ABB RAPID module: qulvOK.mod

MODULE Module1

    CONST robtarget myPath0{255} := [
[[1351.7,1.5,938.01],[0.00139266,-0.491072,0.870802,-0.0234724],[0,-1,-1,0],[9E+09,9E+09,9E+09,9E+09,9E+09,9E+09]],
[[1348.2,2,938.01],[0.00139266,-0.491072,0.870802,-0.0234724],[0,-1,-1,0],[9E+09,9E+09,9E+09,9E+09,9E+09,9E+09]],
[[1346.2,3,938.01],[0.00139266,-0.491072,0.870802,-0.0234724],[0,-1,-1,0],[9E+09,9E+09,9E+09,9E+09,9E+09,9E+09]],
[[1345.7,3,938.01],[0.00139266,-0.491072,0.870802,-0.0234724],[0,-1,-1,0],[9E+09,9E+09,9E+09,9E+09,9E+09,9E+09]],
[[1342.7,5,938.01],[0.00139266,-0.491072,0.870802,-0.0234724],[0,-1,-1,0],[9E+09,9E+09,9E+09,9E+09,9E+09,9E+09]],
[[1340.2,3.5,938.01],[0.00139266,-0.491072,0.870802,-0.0234724],[0,-1,-1,0],[9E+09,9E+09,9E+09,9E+09,9E+09,9E+09]],
[[1339.2,2.5,938.01],[0.00139266,-0.491072,0.870802,-0.0234724],[0,-1,-1,0],[9E+09,9E+09,9E+09,9E+09,9E+09,9E+09]],
[[1336.2,2,938.01],[0.00139266,-0.491072,0.870802,-0.0234724],[0,-1,-1,0],[9E+09,9E+09,9E+09,9E+09,9E+09,9E+09]],
[[1335.7,1.5,938.01],[0.00139266,-0.491072,0.870802,-0.0234724],[0,-1,-1,0],[9E+09,9E+09,9E+09,9E+09,9E+09,9E+09]],
[[1327.7,2,938.01],[0.00139266,-0.491072,0.870802,-0.0234724],[0,-1,-1,0],[9E+09,9E+09,9E+09,9E+09,9E+09,9E+09]],
[[1327.2,2.5,938.01],[0.00139266,-0.491072,0.870802,-0.0234724],[0,-1,-1,0],[9E+09,9E+09,9E+09,9E+09,9E+09,9E+09]],
[[1326.7,2.5,938.01],[0.00139266,-0.491072,0.870802,-0.0234724],[0,-1,-1,0],[9E+09,9E+09,9E+09,9E+09,9E+09,9E+09]],
[[1326.2,3,938.01],[0.00139266,-0.491072,0.870802,-0.0234724],[0,-1,-1,0],[9E+09,9E+09,9E+09,9E+09,9E+09,9E+09]],
[[1319.7,6.5,938.01],[0.00139266,-0.491072,0.870802,-0.0234724],[0,-1,-1,0],[9E+09,9E+09,9E+09,9E+09,9E+09,9E+09]],
[[1319.7,6.5,938.01],[0.00139266,-0.491072,0.870802,-0.0234724],[0,-1,-1,0],[9E+09,9E+09,9E+09,9E+09,9E+09,9E+09]],
[[1319.7,6.5,938.01],[0.00139266,-0.491072,0.870802,-0.0234724],[0,-1,-1,0],[9E+09,9E+09,9E+09,9E+09,9E+09,9E+09]],
[[1319.2,7,938.01],[0.00139266,-0.491072,0.870802,-0.0234724],[0,-1,-1,0],[9E+09,9E+09,9E+09,9E+09,9E+09,9E+09]],
[[1310.2,14.5,938.01],[0.00139266,-0.491072,0.870802,-0.0234724],[0,-1,-1,0],[9E+09,9E+09,9E+09,9E+09,9E+09,9E+09]],
[[1310.2,14.5,938.01],[0.00139266,-0.491072,0.870802,-0.0234724],[0,-1,-1,0],[9E+09,9E+09,9E+09,9E+09,9E+09,9E+09]],
[[1310.2,14.5,938.01],[0.00139266,-0.491072,0.870802,-0.0234724],[0,-1,-1,0],[9E+09,9E+09,9E+09,9E+09,9E+09,9E+09]],
[[1310.2,14.5,938.01],[0.00139266,-0.491072,0.870802,-0.0234724],[0,-1,-1,0],[9E+09,9E+09,9E+09,9E+09,9E+09,9E+09]],
[[1307.2,18.5,938.01],[0.00139266,-0.491072,0.870802,-0.0234724],[0,-1,-1,0],[9E+09,9E+09,9E+09,9E+09,9E+09,9E+09]],
[[1303.7,23,938.01],[0.00139266,-0.491072,0.870802,-0.0234724],[0,-1,-1,0],[9E+09,9E+09,9E+09,9E+09,9E+09,9E+09]],
[[1303.7,22.5,938.01],[0.00139266,-0.491072,0.870802,-0.0234724],[0,-1,-1,0],[9E+09,9E+09,9E+09,9E+09,9E+09,9E+09]],
[[1302.2,25,938.01],[0.00139266,-0.491072,0.870802,-0.0234724],[0,-1,-1,0],[9E+09,9E+09,9E+09,9E+09,9E+09,9E+09]],
[[1302.2,25,938.01],[0.00139266,-0.491072,0.870802,-0.0234724],[0,-1,-1,0],[9E+09,9E+09,9E+09,9E+09,9E+09,9E+09]],
[[1301.7,25.5,938.01],[0.00139266,-0.491072,0.870802,-0.0234724],[0,-1,-1,0],[9E+09,9E+09,9E+09,9E+09,9E+09,9E+09]],
[[1301.7,25.5,938.01],[0.00139266,-0.491072,0.870802,-0.0234724],[0,-1,-1,0],[9E+09,9E+09,9E+09,9E+09,9E+09,9E+09]],
[[1299.7,28.5,938.01],[0.00139266,-0.491072,0.870802,-0.0234724],[0,-1,-1,0],[9E+09,9E+09,9E+09,9E+09,9E+09,9E+09]],
[[1299.7,28.5,938.01],[0.00139266,-0.491072,0.870802,-0.0234724],[0,-1,-1,0],[9E+09,9E+09,9E+09,9E+09,9E+09,9E+09]],
[[1298.7,30,938.01],[0.00139266,-0.491072,0.870802,-0.0234724],[0,-1,-1,0],[9E+09,9E+09,9E+09,9E+09,9E+09,9E+09]],
[[1298.7,30,938.01],[0.00139266,-0.491072,0.870802,-0.0234724],[0,-1,-1,0],[9E+09,9E+09,9E+09,9E+09,9E+09,9E+09]],
[[1297.2,32.5,938.01],[0.00139266,-0.491072,0.870802,-0.0234724],[0,-1,-1,0],[9E+09,9E+09,9E+09,9E+09,9E+09,9E+09]],
[[1295.2,36.5,938.01],[0.00139266,-0.491072,0.870802,-0.0234724],[0,-1,-1,0],[9E+09,9E+09,9E+09,9E+09,9E+09,9E+09]],
[[1295.2,36.5,938.01],[0.00139266,-0.491072,0.870802,-0.0234724],[0,-1,-1,0],[9E+09,9E+09,9E+09,9E+09,9E+09,9E+09]],
[[1294.2,39,938.01],[0.00139266,-0.491072,0.870802,-0.0234724],[0,-1,-1,0],[9E+09,9E+09,9E+09,9E+09,9E+09,9E+09]],
[[1293.7,40,938.01],[0.00139266,-0.491072,0.870802,-0.0234724],[0,-1,-1,0],[9E+09,9E+09,9E+09,9E+09,9E+09,9E+09]],
[[1293.2,41,938.01],[0.00139266,-0.491072,0.870802,-0.0234724],[0,-1,-1,0],[9E+09,9E+09,9E+09,9E+09,9E+09,9E+09]],
[[1293.2,41.5,938.01],[0.00139266,-0.491072,0.870802,-0.0234724],[0,-1,-1,0],[9E+09,9E+09,9E+09,9E+09,9E+09,9E+09]],
[[1292.7,42,938.01],[0.00139266,-0.491072,0.870802,-0.0234724],[0,-1,-1,0],[9E+09,9E+09,9E+09,9E+09,9E+09,9E+09]],
[[1292.7,42.5,938.01],[0.00139266,-0.491072,0.870802,-0.0234724],[0,-1,-1,0],[9E+09,9E+09,9E+09,9E+09,9E+09,9E+09]],
[[1292.7,42.5,938.01],[0.00139266,-0.491072,0.870802,-0.0234724],[0,-1,-1,0],[9E+09,9E+09,9E+09,9E+09,9E+09,9E+09]],
[[1293.2,57,938.01],[0.00139266,-0.491072,0.870802,-0.0234724],[0,-1,-1,0],[9E+09,9E+09,9E+09,9E+09,9E+09,9E+09]],
[[1293.7,58,938.01],[0.00139266,-0.491072,0.870802,-0.0234724],[0,-1,-1,0],[9E+09,9E+09,9E+09,9E+09,9E+09,9E+09]],
[[1293.7,58,938.01],[0.00139266,-0.491072,0.870802,-0.0234724],[0,-1,-1,0],[9E+09,9E+09,9E+09,9E+09,9E+09,9E+09]],
[[1295.7,61,938.01],[0.00139266,-0.491072,0.870802,-0.0234724],[0,-1,-1,0],[9E+09,9E+09,9E+09,9E+09,9E+09,9E+09]],
[[1296.7,62.5,938.01],[0.00139266,-0.491072,0.870802,-0.0234724],[0,-1,-1,0],[9E+09,9E+09,9E+09,9E+09,9E+09,9E+09]],
[[1302.2,67,938.01],[0.00139266,-0.491072,0.870802,-0.0234724],[0,-1,-1,0],[9E+09,9E+09,9E+09,9E+09,9E+09,9E+09]],
[[1302.2,67,938.01],[0.00139266,-0.491072,0.870802,-0.0234724],[0,-1,-1,0],[9E+09,9E+09,9E+09,9E+09,9E+09,9E+09]],
[[1304.2,68.5,938.01],[0.00139266,-0.491072,0.870802,-0.0234724],[0,-1,-1,0],[9E+09,9E+09,9E+09,9E+09,9E+09,9E+09]],
[[1305.2,69,938.01],[0.00139266,-0.491072,0.870802,-0.0234724],[0,-1,-1,0],[9E+09,9E+09,9E+09,9E+09,9E+09,9E+09]],
[[1305.2,69,938.01],[0.00139266,-0.491072,0.870802,-0.0234724],[0,-1,-1,0],[9E+09,9E+09,9E+09,9E+09,9E+09,9E+09]],
[[1307.2,70,938.01],[0.00139266,-0.491072,0.870802,-0.0234724],[0,-1,-1,0],[9E+09,9E+09,9E+09,9E+09,9E+09,9E+09]],
[[1308.7,70,938.01],[0.00139266,-0.491072,0.870802,-0.0234724],[0,-1,-1,0],[9E+09,9E+09,9E+09,9E+09,9E+09,9E+09]],
[[1310.2,72,938.01],[0.00139266,-0.491072,0.870802,-0.0234724],[0,-1,-1,0],[9E+09,9E+09,9E+09,9E+09,9E+09,9E+09]],
[[1313.7,71,938.01],[0.00139266,-0.491072,0.870802,-0.0234724],[0,-1,-1,0],[9E+09,9E+09,9E+09,9E+09,9E+09,9E+09]],
[[1314.2,71.5,938.01],[0.00139266,-0.491072,0.870802,-0.0234724],[0,-1,-1,0],[9E+09,9E+09,9E+09,9E+09,9E+09,9E+09]],
[[1317.7,72,938.01],[0.00139266,-0.491072,0.870802,-0.0234724],[0,-1,-1,0],[9E+09,9E+09,9E+09,9E+09,9E+09,9E+09]],
[[1317.7,72,938.01],[0.00139266,-0.491072,0.870802,-0.0234724],[0,-1,-1,0],[9E+09,9E+09,9E+09,9E+09,9E+09,9E+09]],
[[1317.7,72,938.01],[0.00139266,-0.491072,0.870802,-0.0234724],[0,-1,-1,0],[9E+09,9E+09,9E+09,9E+09,9E+09,9E+09]],
[[1310.2,72,938.01],[0.00139266,-0.491072,0.870802,-0.0234724],[0,-1,-1,0],[9E+09,9E+09,9E+09,9E+09,9E+09,9E+09]],
[[1307.7,73.5,938.01],[0.00139266,-0.491072,0.870802,-0.0234724],[0,-1,-1,0],[9E+09,9E+09,9E+09,9E+09,9E+09,9E+09]],
[[1301.2,74,938.01],[0.00139266,-0.491072,0.870802,-0.0234724],[0,-1,-1,0],[9E+09,9E+09,9E+09,9E+09,9E+09,9E+09]],
[[1300.7,74.5,938.01],[0.00139266,-0.491072,0.870802,-0.0234724],[0,-1,-1,0],[9E+09,9E+09,9E+09,9E+09,9E+09,9E+09]],
[[1299.7,74.5,938.01],[0.00139266,-0.491072,0.870802,-0.0234724],[0,-1,-1,0],[9E+09,9E+09,9E+09,9E+09,9E+09,9E+09]],
[[1299.2,75,938.01],[0.00139266,-0.491072,0.870802,-0.0234724],[0,-1,-1,0],[9E+09,9E+09,9E+09,9E+09,9E+09,9E+09]],
[[1295.7,76,938.01],[0.00139266,-0.491072,0.870802,-0.0234724],[0,-1,-1,0],[9E+09,9E+09,9E+09,9E+09,9E+09,9E+09]],
[[1295.7,76,938.01],[0.00139266,-0.491072,0.870802,-0.0234724],[0,-1,-1,0],[9E+09,9E+09,9E+09,9E+09,9E+09,9E+09]],
[[1295.2,76.5,938.01],[0.00139266,-0.491072,0.870802,-0.0234724],[0,-1,-1,0],[9E+09,9E+09,9E+09,9E+09,9E+09,9E+09]],
[[1294.2,76.5,938.01],[0.00139266,-0.491072,0.870802,-0.0234724],[0,-1,-1,0],[9E+09,9E+09,9E+09,9E+09,9E+09,9E+09]],
[[1292.7,77.5,938.01],[0.00139266,-0.491072,0.870802,-0.0234724],[0,-1,-1,0],[9E+09,9E+09,9E+09,9E+09,9E+09,9E+09]],
[[1292.2,77.5,938.01],[0.00139266,-0.491072,0.870802,-0.0234724],[0,-1,-1,0],[9E+09,9E+09,9E+09,9E+09,9E+09,9E+09]],
[[1292.2,77.5,938.01],[0.00139266,-0.491072,0.870802,-0.0234724],[0,-1,-1,0],[9E+09,9E+09,9E+09,9E+09,9E+09,9E+09]],
[[1286.7,80.5,938.01],[0.00139266,-0.491072,0.870802,-0.0234724],[0,-1,-1,0],[9E+09,9E+09,9E+09,9E+09,9E+09,9E+09]],
[[1286.7,80.5,938.01],[0.00139266,-0.491072,0.870802,-0.0234724],[0,-1,-1,0],[9E+09,9E+09,9E+09,9E+09,9E+09,9E+09]],
[[1286.7,80.5,938.01],[0.00139266,-0.491072,0.870802,-0.0234724],[0,-1,-1,0],[9E+09,9E+09,9E+09,9E+09,9E+09,9E+09]],
[[1280.7,75,938.01],[0.00139266,-0.491072,0.870802,-0.0234724],[0,-1,-1,0],[9E+09,9E+09,9E+09,9E+09,9E+09,9E+09]],
[[1281.2,68.5,938.01],[0.00139266,-0.491072,0.870802,-0.0234724],[0,-1,-1,0],[9E+09,9E+09,9E+09,9E+09,9E+09,9E+09]],
[[1281.2,68.5,938.01],[0.00139266,-0.491072,0.870802,-0.0234724],[0,-1,-1,0],[9E+09,9E+09,9E+09,9E+09,9E+09,9E+09]],
[[1282.7,66.5,938.01],[0.00139266,-0.491072,0.870802,-0.0234724],[0,-1,-1,0],[9E+09,9E+09,9E+09,9E+09,9E+09,9E+09]],
[[1282.7,66,938.01],[0.00139266,-0.491072,0.870802,-0.0234724],[0,-1,-1,0],[9E+09,9E+09,9E+09,9E+09,9E+09,9E+09]],
[[1280.7,63,938.01],[0.00139266,-0.491072,0.870802,-0.0234724],[0,-1,-1,0],[9E+09,9E+09,9E+09,9E+09,9E+09,9E+09]],
[[1280.2,63.5,938.01],[0.00139266,-0.491072,0.870802,-0.0234724],[0,-1,-1,0],[9E+09,9E+09,9E+09,9E+09,9E+09,9E+09]],
[[1279.7,63.5,938.01],[0.00139266,-0.491072,0.870802,-0.0234724],[0,-1,-1,0],[9E+09,9E+09,9E+09,9E+09,9E+09,9E+09]],
[[1278.2,64,938.01],[0.00139266,-0.491072,0.870802,-0.0234724],[0,-1,-1,0],[9E+09,9E+09,9E+09,9E+09,9E+09,9E+09]],
[[1277.7,64,938.01],[0.00139266,-0.491072,0.870802,-0.0234724],[0,-1,-1,0],[9E+09,9E+09,9E+09,9E+09,9E+09,9E+09]],
[[1276.7,64.5,938.01],[0.00139266,-0.491072,0.870802,-0.0234724],[0,-1,-1,0],[9E+09,9E+09,9E+09,9E+09,9E+09,9E+09]],
[[1276.2,64.5,938.01],[0.00139266,-0.491072,0.870802,-0.0234724],[0,-1,-1,0],[9E+09,9E+09,9E+09,9E+09,9E+09,9E+09]],
[[1275.7,65,938.01],[0.00139266,-0.491072,0.870802,-0.0234724],[0,-1,-1,0],[9E+09,9E+09,9E+09,9E+09,9E+09,9E+09]],
[[1275.7,65,938.01],[0.00139266,-0.491072,0.870802,-0.0234724],[0,-1,-1,0],[9E+09,9E+09,9E+09,9E+09,9E+09,9E+09]],
[[1274.2,66,938.01],[0.00139266,-0.491072,0.870802,-0.0234724],[0,-1,-1,0],[9E+09,9E+09,9E+09,9E+09,9E+09,9E+09]],
[[1273.2,66,938.01],[0.00139266,-0.491072,0.870802,-0.0234724],[0,-1,-1,0],[9E+09,9E+09,9E+09,9E+09,9E+09,9E+09]],
[[1266.2,74,938.01],[0.00139266,-0.491072,0.870802,-0.0234724],[0,-1,-1,0],[9E+09,9E+09,9E+09,9E+09,9E+09,9E+09]],
[[1266.2,74,938.01],[0.00139266,-0.491072,0.870802,-0.0234724],[0,-1,-1,0],[9E+09,9E+09,9E+09,9E+09,9E+09,9E+09]],
[[1266.2,74,938.01],[0.00139266,-0.491072,0.870802,-0.0234724],[0,-1,-1,0],[9E+09,9E+09,9E+09,9E+09,9E+09,9E+09]],
[[1266.2,74,938.01],[0.00139266,-0.491072,0.870802,-0.0234724],[0,-1,-1,0],[9E+09,9E+09,9E+09,9E+09,9E+09,9E+09]],
[[1266.2,74,938.01],[0.00139266,-0.491072,0.870802,-0.0234724],[0,-1,-1,0],[9E+09,9E+09,9E+09,9E+09,9E+09,9E+09]],
[[1266.2,84,938.01],[0.00139266,-0.491072,0.870802,-0.0234724],[0,-1,-1,0],[9E+09,9E+09,9E+09,9E+09,9E+09,9E+09]],
[[1266.7,85,938.01],[0.00139266,-0.491072,0.870802,-0.0234724],[0,-1,-1,0],[9E+09,9E+09,9E+09,9E+09,9E+09,9E+09]],
[[1270.7,88.5,938.01],[0.00139266,-0.491072,0.870802,-0.0234724],[0,-1,-1,0],[9E+09,9E+09,9E+09,9E+09,9E+09,9E+09]],
[[1274.7,89.5,938.01],[0.00139266,-0.491072,0.870802,-0.0234724],[0,-1,-1,0],[9E+09,9E+09,9E+09,9E+09,9E+09,9E+09]],
[[1275.2,90,938.01],[0.00139266,-0.491072,0.870802,-0.0234724],[0,-1,-1,0],[9E+09,9E+09,9E+09,9E+09,9E+09,9E+09]],
[[1279.2,92.5,938.01],[0.00139266,-0.491072,0.870802,-0.0234724],[0,-1,-1,0],[9E+09,9E+09,9E+09,9E+09,9E+09,9E+09]],
[[1278.7,93,938.01],[0.00139266,-0.491072,0.870802,-0.0234724],[0,-1,-1,0],[9E+09,9E+09,9E+09,9E+09,9E+09,9E+09]],
[[1278.7,94,938.01],[0.00139266,-0.491072,0.870802,-0.0234724],[0,-1,-1,0],[9E+09,9E+09,9E+09,9E+09,9E+09,9E+09]],
[[1278.2,94.5,938.01],[0.00139266,-0.491072,0.870802,-0.0234724],[0,-1,-1,0],[9E+09,9E+09,9E+09,9E+09,9E+09,9E+09]],
[[1278.7,106,938.01],[0.00139266,-0.491072,0.870802,-0.0234724],[0,-1,-1,0],[9E+09,9E+09,9E+09,9E+09,9E+09,9E+09]],
[[1279.2,108,938.01],[0.00139266,-0.491072,0.870802,-0.0234724],[0,-1,-1,0],[9E+09,9E+09,9E+09,9E+09,9E+09,9E+09]],
[[1279.7,109,938.01],[0.00139266,-0.491072,0.870802,-0.0234724],[0,-1,-1,0],[9E+09,9E+09,9E+09,9E+09,9E+09,9E+09]],
[[1280.2,110.5,938.01],[0.00139266,-0.491072,0.870802,-0.0234724],[0,-1,-1,0],[9E+09,9E+09,9E+09,9E+09,9E+09,9E+09]],
[[1280.2,110.5,938.01],[0.00139266,-0.491072,0.870802,-0.0234724],[0,-1,-1,0],[9E+09,9E+09,9E+09,9E+09,9E+09,9E+09]],
[[1280.7,111,938.01],[0.00139266,-0.491072,0.870802,-0.0234724],[0,-1,-1,0],[9E+09,9E+09,9E+09,9E+09,9E+09,9E+09]],
[[1280.7,111,938.01],[0.00139266,-0.491072,0.870802,-0.0234724],[0,-1,-1,0],[9E+09,9E+09,9E+09,9E+09,9E+09,9E+09]],
[[1285.7,117.5,938.01],[0.00139266,-0.491072,0.870802,-0.0234724],[0,-1,-1,0],[9E+09,9E+09,9E+09,9E+09,9E+09,9E+09]],
[[1285.7,118,938.01],[0.00139266,-0.491072,0.870802,-0.0234724],[0,-1,-1,0],[9E+09,9E+09,9E+09,9E+09,9E+09,9E+09]],
[[1286.2,118,938.01],[0.00139266,-0.491072,0.870802,-0.0234724],[0,-1,-1,0],[9E+09,9E+09,9E+09,9E+09,9E+09,9E+09]],
[[1287.2,119,938.01],[0.00139266,-0.491072,0.870802,-0.0234724],[0,-1,-1,0],[9E+09,9E+09,9E+09,9E+09,9E+09,9E+09]],
[[1288.2,119.5,938.01],[0.00139266,-0.491072,0.870802,-0.0234724],[0,-1,-1,0],[9E+09,9E+09,9E+09,9E+09,9E+09,9E+09]],
[[1290.2,120.5,938.01],[0.00139266,-0.491072,0.870802,-0.0234724],[0,-1,-1,0],[9E+09,9E+09,9E+09,9E+09,9E+09,9E+09]],
[[1291.7,121.5,938.01],[0.00139266,-0.491072,0.870802,-0.0234724],[0,-1,-1,0],[9E+09,9E+09,9E+09,9E+09,9E+09,9E+09]],
[[1292.2,121.5,938.01],[0.00139266,-0.491072,0.870802,-0.0234724],[0,-1,-1,0],[9E+09,9E+09,9E+09,9E+09,9E+09,9E+09]],
[[1292.2,121.5,938.01],[0.00139266,-0.491072,0.870802,-0.0234724],[0,-1,-1,0],[9E+09,9E+09,9E+09,9E+09,9E+09,9E+09]],
[[1301.2,121.5,938.01],[0.00139266,-0.491072,0.870802,-0.0234724],[0,-1,-1,0],[9E+09,9E+09,9E+09,9E+09,9E+09,9E+09]],
[[1301.7,121,938.01],[0.00139266,-0.491072,0.870802,-0.0234724],[0,-1,-1,0],[9E+09,9E+09,9E+09,9E+09,9E+09,9E+09]],
[[1302.7,121,938.01],[0.00139266,-0.491072,0.870802,-0.0234724],[0,-1,-1,0],[9E+09,9E+09,9E+09,9E+09,9E+09,9E+09]],
[[1303.2,120.5,938.01],[0.00139266,-0.491072,0.870802,-0.0234724],[0,-1,-1,0],[9E+09,9E+09,9E+09,9E+09,9E+09,9E+09]],
[[1306.2,119.5,938.01],[0.00139266,-0.491072,0.870802,-0.0234724],[0,-1,-1,0],[9E+09,9E+09,9E+09,9E+09,9E+09,9E+09]],
[[1306.2,119.5,938.01],[0.00139266,-0.491072,0.870802,-0.0234724],[0,-1,-1,0],[9E+09,9E+09,9E+09,9E+09,9E+09,9E+09]],
[[1308.7,119.5,938.01],[0.00139266,-0.491072,0.870802,-0.0234724],[0,-1,-1,0],[9E+09,9E+09,9E+09,9E+09,9E+09,9E+09]],
[[1309.2,119,938.01],[0.00139266,-0.491072,0.870802,-0.0234724],[0,-1,-1,0],[9E+09,9E+09,9E+09,9E+09,9E+09,9E+09]],
[[1310.7,119,938.01],[0.00139266,-0.491072,0.870802,-0.0234724],[0,-1,-1,0],[9E+09,9E+09,9E+09,9E+09,9E+09,9E+09]],
[[1311.2,118.5,938.01],[0.00139266,-0.491072,0.870802,-0.0234724],[0,-1,-1,0],[9E+09,9E+09,9E+09,9E+09,9E+09,9E+09]],
[[1311.7,118.5,938.01],[0.00139266,-0.491072,0.870802,-0.0234724],[0,-1,-1,0],[9E+09,9E+09,9E+09,9E+09,9E+09,9E+09]],
[[1312.7,117.5,938.01],[0.00139266,-0.491072,0.870802,-0.0234724],[0,-1,-1,0],[9E+09,9E+09,9E+09,9E+09,9E+09,9E+09]],
[[1312.7,116.5,938.01],[0.00139266,-0.491072,0.870802,-0.0234724],[0,-1,-1,0],[9E+09,9E+09,9E+09,9E+09,9E+09,9E+09]],
[[1312.2,116,938.01],[0.00139266,-0.491072,0.870802,-0.0234724],[0,-1,-1,0],[9E+09,9E+09,9E+09,9E+09,9E+09,9E+09]],
[[1312.2,115.5,938.01],[0.00139266,-0.491072,0.870802,-0.0234724],[0,-1,-1,0],[9E+09,9E+09,9E+09,9E+09,9E+09,9E+09]],
[[1311.7,115,938.01],[0.00139266,-0.491072,0.870802,-0.0234724],[0,-1,-1,0],[9E+09,9E+09,9E+09,9E+09,9E+09,9E+09]],
[[1311.7,114,938.01],[0.00139266,-0.491072,0.870802,-0.0234724],[0,-1,-1,0],[9E+09,9E+09,9E+09,9E+09,9E+09,9E+09]],
[[1312.2,113.5,938.01],[0.00139266,-0.491072,0.870802,-0.0234724],[0,-1,-1,0],[9E+09,9E+09,9E+09,9E+09,9E+09,9E+09]],
[[1313.2,113.5,938.01],[0.00139266,-0.491072,0.870802,-0.0234724],[0,-1,-1,0],[9E+09,9E+09,9E+09,9E+09,9E+09,9E+09]],
[[1313.7,114,938.01],[0.00139266,-0.491072,0.870802,-0.0234724],[0,-1,-1,0],[9E+09,9E+09,9E+09,9E+09,9E+09,9E+09]],
[[1320.2,114,938.01],[0.00139266,-0.491072,0.870802,-0.0234724],[0,-1,-1,0],[9E+09,9E+09,9E+09,9E+09,9E+09,9E+09]],
[[1325.2,120,938.01],[0.00139266,-0.491072,0.870802,-0.0234724],[0,-1,-1,0],[9E+09,9E+09,9E+09,9E+09,9E+09,9E+09]],
[[1325.2,120,938.01],[0.00139266,-0.491072,0.870802,-0.0234724],[0,-1,-1,0],[9E+09,9E+09,9E+09,9E+09,9E+09,9E+09]],
[[1326.2,120.5,938.01],[0.00139266,-0.491072,0.870802,-0.0234724],[0,-1,-1,0],[9E+09,9E+09,9E+09,9E+09,9E+09,9E+09]],
[[1341.2,121.5,938.01],[0.00139266,-0.491072,0.870802,-0.0234724],[0,-1,-1,0],[9E+09,9E+09,9E+09,9E+09,9E+09,9E+09]],
[[1341.7,121,938.01],[0.00139266,-0.491072,0.870802,-0.0234724],[0,-1,-1,0],[9E+09,9E+09,9E+09,9E+09,9E+09,9E+09]],
[[1342.7,121,938.01],[0.00139266,-0.491072,0.870802,-0.0234724],[0,-1,-1,0],[9E+09,9E+09,9E+09,9E+09,9E+09,9E+09]],
[[1343.2,120.5,938.01],[0.00139266,-0.491072,0.870802,-0.0234724],[0,-1,-1,0],[9E+09,9E+09,9E+09,9E+09,9E+09,9E+09]],
[[1343.7,113.5,938.01],[0.00139266,-0.491072,0.870802,-0.0234724],[0,-1,-1,0],[9E+09,9E+09,9E+09,9E+09,9E+09,9E+09]],
[[1343.7,113.5,938.01],[0.00139266,-0.491072,0.870802,-0.0234724],[0,-1,-1,0],[9E+09,9E+09,9E+09,9E+09,9E+09,9E+09]],
[[1343.7,113.5,938.01],[0.00139266,-0.491072,0.870802,-0.0234724],[0,-1,-1,0],[9E+09,9E+09,9E+09,9E+09,9E+09,9E+09]],
[[1343.7,113.5,938.01],[0.00139266,-0.491072,0.870802,-0.0234724],[0,-1,-1,0],[9E+09,9E+09,9E+09,9E+09,9E+09,9E+09]],
[[1346.7,113,938.01],[0.00139266,-0.491072,0.870802,-0.0234724],[0,-1,-1,0],[9E+09,9E+09,9E+09,9E+09,9E+09,9E+09]],
[[1347.2,112.5,938.01],[0.00139266,-0.491072,0.870802,-0.0234724],[0,-1,-1,0],[9E+09,9E+09,9E+09,9E+09,9E+09,9E+09]],
[[1348.7,112.5,938.01],[0.00139266,-0.491072,0.870802,-0.0234724],[0,-1,-1,0],[9E+09,9E+09,9E+09,9E+09,9E+09,9E+09]],
[[1349.2,112,938.01],[0.00139266,-0.491072,0.870802,-0.0234724],[0,-1,-1,0],[9E+09,9E+09,9E+09,9E+09,9E+09,9E+09]],
[[1352.7,111,938.01],[0.00139266,-0.491072,0.870802,-0.0234724],[0,-1,-1,0],[9E+09,9E+09,9E+09,9E+09,9E+09,9E+09]],
[[1352.7,111,938.01],[0.00139266,-0.491072,0.870802,-0.0234724],[0,-1,-1,0],[9E+09,9E+09,9E+09,9E+09,9E+09,9E+09]],
[[1352.7,111,938.01],[0.00139266,-0.491072,0.870802,-0.0234724],[0,-1,-1,0],[9E+09,9E+09,9E+09,9E+09,9E+09,9E+09]],
[[1356.7,108,938.01],[0.00139266,-0.491072,0.870802,-0.0234724],[0,-1,-1,0],[9E+09,9E+09,9E+09,9E+09,9E+09,9E+09]],
[[1356.2,105,938.01],[0.00139266,-0.491072,0.870802,-0.0234724],[0,-1,-1,0],[9E+09,9E+09,9E+09,9E+09,9E+09,9E+09]],
[[1356.2,105,938.01],[0.00139266,-0.491072,0.870802,-0.0234724],[0,-1,-1,0],[9E+09,9E+09,9E+09,9E+09,9E+09,9E+09]],
[[1353.2,102.5,938.01],[0.00139266,-0.491072,0.870802,-0.0234724],[0,-1,-1,0],[9E+09,9E+09,9E+09,9E+09,9E+09,9E+09]],
[[1353.2,102.5,938.01],[0.00139266,-0.491072,0.870802,-0.0234724],[0,-1,-1,0],[9E+09,9E+09,9E+09,9E+09,9E+09,9E+09]],
[[1353.2,102.5,938.01],[0.00139266,-0.491072,0.870802,-0.0234724],[0,-1,-1,0],[9E+09,9E+09,9E+09,9E+09,9E+09,9E+09]],
[[1352.7,99,938.01],[0.00139266,-0.491072,0.870802,-0.0234724],[0,-1,-1,0],[9E+09,9E+09,9E+09,9E+09,9E+09,9E+09]],
[[1352.2,98.5,938.01],[0.00139266,-0.491072,0.870802,-0.0234724],[0,-1,-1,0],[9E+09,9E+09,9E+09,9E+09,9E+09,9E+09]],
[[1352.2,97.5,938.01],[0.00139266,-0.491072,0.870802,-0.0234724],[0,-1,-1,0],[9E+09,9E+09,9E+09,9E+09,9E+09,9E+09]],
[[1350.7,95,938.01],[0.00139266,-0.491072,0.870802,-0.0234724],[0,-1,-1,0],[9E+09,9E+09,9E+09,9E+09,9E+09,9E+09]],
[[1350.7,95,938.01],[0.00139266,-0.491072,0.870802,-0.0234724],[0,-1,-1,0],[9E+09,9E+09,9E+09,9E+09,9E+09,9E+09]],
[[1350.7,95,938.01],[0.00139266,-0.491072,0.870802,-0.0234724],[0,-1,-1,0],[9E+09,9E+09,9E+09,9E+09,9E+09,9E+09]],
[[1352.2,89,938.01],[0.00139266,-0.491072,0.870802,-0.0234724],[0,-1,-1,0],[9E+09,9E+09,9E+09,9E+09,9E+09,9E+09]],
[[1350.7,86.5,938.01],[0.00139266,-0.491072,0.870802,-0.0234724],[0,-1,-1,0],[9E+09,9E+09,9E+09,9E+09,9E+09,9E+09]],
[[1352.7,83.5,938.01],[0.00139266,-0.491072,0.870802,-0.0234724],[0,-1,-1,0],[9E+09,9E+09,9E+09,9E+09,9E+09,9E+09]],
[[1353.7,81,938.01],[0.00139266,-0.491072,0.870802,-0.0234724],[0,-1,-1,0],[9E+09,9E+09,9E+09,9E+09,9E+09,9E+09]],
[[1353.7,81,938.01],[0.00139266,-0.491072,0.870802,-0.0234724],[0,-1,-1,0],[9E+09,9E+09,9E+09,9E+09,9E+09,9E+09]],
[[1368.2,78.5,938.01],[0.00139266,-0.491072,0.870802,-0.0234724],[0,-1,-1,0],[9E+09,9E+09,9E+09,9E+09,9E+09,9E+09]],
[[1368.2,78.5,938.01],[0.00139266,-0.491072,0.870802,-0.0234724],[0,-1,-1,0],[9E+09,9E+09,9E+09,9E+09,9E+09,9E+09]],
[[1368.2,78.5,938.01],[0.00139266,-0.491072,0.870802,-0.0234724],[0,-1,-1,0],[9E+09,9E+09,9E+09,9E+09,9E+09,9E+09]],
[[1368.2,78.5,938.01],[0.00139266,-0.491072,0.870802,-0.0234724],[0,-1,-1,0],[9E+09,9E+09,9E+09,9E+09,9E+09,9E+09]],
[[1368.2,78,938.01],[0.00139266,-0.491072,0.870802,-0.0234724],[0,-1,-1,0],[9E+09,9E+09,9E+09,9E+09,9E+09,9E+09]],
[[1370.2,77.5,938.01],[0.00139266,-0.491072,0.870802,-0.0234724],[0,-1,-1,0],[9E+09,9E+09,9E+09,9E+09,9E+09,9E+09]],
[[1371.2,77.5,938.01],[0.00139266,-0.491072,0.870802,-0.0234724],[0,-1,-1,0],[9E+09,9E+09,9E+09,9E+09,9E+09,9E+09]],
[[1371.7,77,938.01],[0.00139266,-0.491072,0.870802,-0.0234724],[0,-1,-1,0],[9E+09,9E+09,9E+09,9E+09,9E+09,9E+09]],
[[1372.2,77,938.01],[0.00139266,-0.491072,0.870802,-0.0234724],[0,-1,-1,0],[9E+09,9E+09,9E+09,9E+09,9E+09,9E+09]],
[[1373.7,76.5,938.01],[0.00139266,-0.491072,0.870802,-0.0234724],[0,-1,-1,0],[9E+09,9E+09,9E+09,9E+09,9E+09,9E+09]],
[[1374.2,76.5,938.01],[0.00139266,-0.491072,0.870802,-0.0234724],[0,-1,-1,0],[9E+09,9E+09,9E+09,9E+09,9E+09,9E+09]],
[[1374.7,76,938.01],[0.00139266,-0.491072,0.870802,-0.0234724],[0,-1,-1,0],[9E+09,9E+09,9E+09,9E+09,9E+09,9E+09]],
[[1375.2,76,938.01],[0.00139266,-0.491072,0.870802,-0.0234724],[0,-1,-1,0],[9E+09,9E+09,9E+09,9E+09,9E+09,9E+09]],
[[1375.7,76,938.01],[0.00139266,-0.491072,0.870802,-0.0234724],[0,-1,-1,0],[9E+09,9E+09,9E+09,9E+09,9E+09,9E+09]],
[[1376.2,75.5,938.01],[0.00139266,-0.491072,0.870802,-0.0234724],[0,-1,-1,0],[9E+09,9E+09,9E+09,9E+09,9E+09,9E+09]],
[[1377.2,75,938.01],[0.00139266,-0.491072,0.870802,-0.0234724],[0,-1,-1,0],[9E+09,9E+09,9E+09,9E+09,9E+09,9E+09]],
[[1377.2,75,938.01],[0.00139266,-0.491072,0.870802,-0.0234724],[0,-1,-1,0],[9E+09,9E+09,9E+09,9E+09,9E+09,9E+09]],
[[1379.2,74,938.01],[0.00139266,-0.491072,0.870802,-0.0234724],[0,-1,-1,0],[9E+09,9E+09,9E+09,9E+09,9E+09,9E+09]],
[[1379.2,74,938.01],[0.00139266,-0.491072,0.870802,-0.0234724],[0,-1,-1,0],[9E+09,9E+09,9E+09,9E+09,9E+09,9E+09]],
[[1381.7,72.5,938.01],[0.00139266,-0.491072,0.870802,-0.0234724],[0,-1,-1,0],[9E+09,9E+09,9E+09,9E+09,9E+09,9E+09]],
[[1384.2,71,938.01],[0.00139266,-0.491072,0.870802,-0.0234724],[0,-1,-1,0],[9E+09,9E+09,9E+09,9E+09,9E+09,9E+09]],
[[1384.2,71,938.01],[0.00139266,-0.491072,0.870802,-0.0234724],[0,-1,-1,0],[9E+09,9E+09,9E+09,9E+09,9E+09,9E+09]],
[[1384.2,71,938.01],[0.00139266,-0.491072,0.870802,-0.0234724],[0,-1,-1,0],[9E+09,9E+09,9E+09,9E+09,9E+09,9E+09]],
[[1384.2,71,938.01],[0.00139266,-0.491072,0.870802,-0.0234724],[0,-1,-1,0],[9E+09,9E+09,9E+09,9E+09,9E+09,9E+09]],
[[1385.2,70.5,938.01],[0.00139266,-0.491072,0.870802,-0.0234724],[0,-1,-1,0],[9E+09,9E+09,9E+09,9E+09,9E+09,9E+09]],
[[1386.2,69.5,938.01],[0.00139266,-0.491072,0.870802,-0.0234724],[0,-1,-1,0],[9E+09,9E+09,9E+09,9E+09,9E+09,9E+09]],
[[1388.7,67.5,938.01],[0.00139266,-0.491072,0.870802,-0.0234724],[0,-1,-1,0],[9E+09,9E+09,9E+09,9E+09,9E+09,9E+09]],
[[1392.7,63.5,938.01],[0.00139266,-0.491072,0.870802,-0.0234724],[0,-1,-1,0],[9E+09,9E+09,9E+09,9E+09,9E+09,9E+09]],
[[1393.2,63,938.01],[0.00139266,-0.491072,0.870802,-0.0234724],[0,-1,-1,0],[9E+09,9E+09,9E+09,9E+09,9E+09,9E+09]],
[[1395.2,60,938.01],[0.00139266,-0.491072,0.870802,-0.0234724],[0,-1,-1,0],[9E+09,9E+09,9E+09,9E+09,9E+09,9E+09]],
[[1395.7,59,938.01],[0.00139266,-0.491072,0.870802,-0.0234724],[0,-1,-1,0],[9E+09,9E+09,9E+09,9E+09,9E+09,9E+09]],
[[1396.2,58.5,938.01],[0.00139266,-0.491072,0.870802,-0.0234724],[0,-1,-1,0],[9E+09,9E+09,9E+09,9E+09,9E+09,9E+09]],
[[1396.7,57.5,938.01],[0.00139266,-0.491072,0.870802,-0.0234724],[0,-1,-1,0],[9E+09,9E+09,9E+09,9E+09,9E+09,9E+09]],
[[1397.2,56.5,938.01],[0.00139266,-0.491072,0.870802,-0.0234724],[0,-1,-1,0],[9E+09,9E+09,9E+09,9E+09,9E+09,9E+09]],
[[1397.7,56,938.01],[0.00139266,-0.491072,0.870802,-0.0234724],[0,-1,-1,0],[9E+09,9E+09,9E+09,9E+09,9E+09,9E+09]],
[[1397.7,56,938.01],[0.00139266,-0.491072,0.870802,-0.0234724],[0,-1,-1,0],[9E+09,9E+09,9E+09,9E+09,9E+09,9E+09]],
[[1398.2,52.5,938.01],[0.00139266,-0.491072,0.870802,-0.0234724],[0,-1,-1,0],[9E+09,9E+09,9E+09,9E+09,9E+09,9E+09]],
[[1398.7,51,938.01],[0.00139266,-0.491072,0.870802,-0.0234724],[0,-1,-1,0],[9E+09,9E+09,9E+09,9E+09,9E+09,9E+09]],
[[1397.7,44.5,938.01],[0.00139266,-0.491072,0.870802,-0.0234724],[0,-1,-1,0],[9E+09,9E+09,9E+09,9E+09,9E+09,9E+09]],
[[1397.7,44.5,938.01],[0.00139266,-0.491072,0.870802,-0.0234724],[0,-1,-1,0],[9E+09,9E+09,9E+09,9E+09,9E+09,9E+09]],
[[1397.7,44.5,938.01],[0.00139266,-0.491072,0.870802,-0.0234724],[0,-1,-1,0],[9E+09,9E+09,9E+09,9E+09,9E+09,9E+09]],
[[1400.7,42.5,938.01],[0.00139266,-0.491072,0.870802,-0.0234724],[0,-1,-1,0],[9E+09,9E+09,9E+09,9E+09,9E+09,9E+09]],
[[1400.7,42.5,938.01],[0.00139266,-0.491072,0.870802,-0.0234724],[0,-1,-1,0],[9E+09,9E+09,9E+09,9E+09,9E+09,9E+09]],
[[1401.2,41.5,938.01],[0.00139266,-0.491072,0.870802,-0.0234724],[0,-1,-1,0],[9E+09,9E+09,9E+09,9E+09,9E+09,9E+09]],
[[1401.2,35.5,938.01],[0.00139266,-0.491072,0.870802,-0.0234724],[0,-1,-1,0],[9E+09,9E+09,9E+09,9E+09,9E+09,9E+09]],
[[1401.2,35.5,938.01],[0.00139266,-0.491072,0.870802,-0.0234724],[0,-1,-1,0],[9E+09,9E+09,9E+09,9E+09,9E+09,9E+09]],
[[1400.7,34.5,938.01],[0.00139266,-0.491072,0.870802,-0.0234724],[0,-1,-1,0],[9E+09,9E+09,9E+09,9E+09,9E+09,9E+09]],
[[1396.7,31.5,938.01],[0.00139266,-0.491072,0.870802,-0.0234724],[0,-1,-1,0],[9E+09,9E+09,9E+09,9E+09,9E+09,9E+09]],
[[1396.7,31.5,938.01],[0.00139266,-0.491072,0.870802,-0.0234724],[0,-1,-1,0],[9E+09,9E+09,9E+09,9E+09,9E+09,9E+09]],
[[1396.7,31.5,938.01],[0.00139266,-0.491072,0.870802,-0.0234724],[0,-1,-1,0],[9E+09,9E+09,9E+09,9E+09,9E+09,9E+09]],
[[1396.2,31.5,938.01],[0.00139266,-0.491072,0.870802,-0.0234724],[0,-1,-1,0],[9E+09,9E+09,9E+09,9E+09,9E+09,9E+09]],
[[1396.2,31.5,938.01],[0.00139266,-0.491072,0.870802,-0.0234724],[0,-1,-1,0],[9E+09,9E+09,9E+09,9E+09,9E+09,9E+09]],
[[1390.2,30.5,938.01],[0.00139266,-0.491072,0.870802,-0.0234724],[0,-1,-1,0],[9E+09,9E+09,9E+09,9E+09,9E+09,9E+09]],
[[1390.2,30.5,938.01],[0.00139266,-0.491072,0.870802,-0.0234724],[0,-1,-1,0],[9E+09,9E+09,9E+09,9E+09,9E+09,9E+09]],
[[1385.2,25,938.01],[0.00139266,-0.491072,0.870802,-0.0234724],[0,-1,-1,0],[9E+09,9E+09,9E+09,9E+09,9E+09,9E+09]],
[[1384.7,24.5,938.01],[0.00139266,-0.491072,0.870802,-0.0234724],[0,-1,-1,0],[9E+09,9E+09,9E+09,9E+09,9E+09,9E+09]],
[[1384.7,24.5,938.01],[0.00139266,-0.491072,0.870802,-0.0234724],[0,-1,-1,0],[9E+09,9E+09,9E+09,9E+09,9E+09,9E+09]],
[[1384.2,24,938.01],[0.00139266,-0.491072,0.870802,-0.0234724],[0,-1,-1,0],[9E+09,9E+09,9E+09,9E+09,9E+09,9E+09]],
[[1381.7,20.5,938.01],[0.00139266,-0.491072,0.870802,-0.0234724],[0,-1,-1,0],[9E+09,9E+09,9E+09,9E+09,9E+09,9E+09]],
[[1381.2,19.5,938.01],[0.00139266,-0.491072,0.870802,-0.0234724],[0,-1,-1,0],[9E+09,9E+09,9E+09,9E+09,9E+09,9E+09]],
[[1380.7,19,938.01],[0.00139266,-0.491072,0.870802,-0.0234724],[0,-1,-1,0],[9E+09,9E+09,9E+09,9E+09,9E+09,9E+09]],
[[1380.7,19,938.01],[0.00139266,-0.491072,0.870802,-0.0234724],[0,-1,-1,0],[9E+09,9E+09,9E+09,9E+09,9E+09,9E+09]],
[[1377.7,15,938.01],[0.00139266,-0.491072,0.870802,-0.0234724],[0,-1,-1,0],[9E+09,9E+09,9E+09,9E+09,9E+09,9E+09]],
[[1376.7,13.5,938.01],[0.00139266,-0.491072,0.870802,-0.0234724],[0,-1,-1,0],[9E+09,9E+09,9E+09,9E+09,9E+09,9E+09]],
[[1371.2,7.5,938.01],[0.00139266,-0.491072,0.870802,-0.0234724],[0,-1,-1,0],[9E+09,9E+09,9E+09,9E+09,9E+09,9E+09]],
[[1370.7,7.5,938.01],[0.00139266,-0.491072,0.870802,-0.0234724],[0,-1,-1,0],[9E+09,9E+09,9E+09,9E+09,9E+09,9E+09]],
[[1367.2,5,938.01],[0.00139266,-0.491072,0.870802,-0.0234724],[0,-1,-1,0],[9E+09,9E+09,9E+09,9E+09,9E+09,9E+09]],
[[1367.2,5,938.01],[0.00139266,-0.491072,0.870802,-0.0234724],[0,-1,-1,0],[9E+09,9E+09,9E+09,9E+09,9E+09,9E+09]],
[[1366.7,4.5,938.01],[0.00139266,-0.491072,0.870802,-0.0234724],[0,-1,-1,0],[9E+09,9E+09,9E+09,9E+09,9E+09,9E+09]],
[[1366.2,4.5,938.01],[0.00139266,-0.491072,0.870802,-0.0234724],[0,-1,-1,0],[9E+09,9E+09,9E+09,9E+09,9E+09,9E+09]],
[[1365.2,4,938.01],[0.00139266,-0.491072,0.870802,-0.0234724],[0,-1,-1,0],[9E+09,9E+09,9E+09,9E+09,9E+09,9E+09]],
[[1364.7,3.5,938.01],[0.00139266,-0.491072,0.870802,-0.0234724],[0,-1,-1,0],[9E+09,9E+09,9E+09,9E+09,9E+09,9E+09]],
[[1363.7,3,938.01],[0.00139266,-0.491072,0.870802,-0.0234724],[0,-1,-1,0],[9E+09,9E+09,9E+09,9E+09,9E+09,9E+09]],
[[1362.7,2.5,938.01],[0.00139266,-0.491072,0.870802,-0.0234724],[0,-1,-1,0],[9E+09,9E+09,9E+09,9E+09,9E+09,9E+09]],
[[1361.7,2,938.01],[0.00139266,-0.491072,0.870802,-0.0234724],[0,-1,-1,0],[9E+09,9E+09,9E+09,9E+09,9E+09,9E+09]],
[[1358.2,1.5,938.01],[0.00139266,-0.491072,0.870802,-0.0234724],[0,-1,-1,0],[9E+09,9E+09,9E+09,9E+09,9E+09,9E+09]],
[[1358.7,1.5,938.01],[0.00139266,-0.491072,0.870802,-0.0234724],[0,-1,-1,0],[9E+09,9E+09,9E+09,9E+09,9E+09,9E+09]]
];
CONST robtarget myPath1{15} := [
[[1311.7,115,938.01],[0.00139266,-0.491072,0.870802,-0.0234724],[0,-1,-1,0],[9E+09,9E+09,9E+09,9E+09,9E+09,9E+09]],
[[1312.2,115.5,938.01],[0.00139266,-0.491072,0.870802,-0.0234724],[0,-1,-1,0],[9E+09,9E+09,9E+09,9E+09,9E+09,9E+09]],
[[1312.2,116,938.01],[0.00139266,-0.491072,0.870802,-0.0234724],[0,-1,-1,0],[9E+09,9E+09,9E+09,9E+09,9E+09,9E+09]],
[[1312.7,116.5,938.01],[0.00139266,-0.491072,0.870802,-0.0234724],[0,-1,-1,0],[9E+09,9E+09,9E+09,9E+09,9E+09,9E+09]],
[[1312.7,117.5,938.01],[0.00139266,-0.491072,0.870802,-0.0234724],[0,-1,-1,0],[9E+09,9E+09,9E+09,9E+09,9E+09,9E+09]],
[[1311.7,118.5,938.01],[0.00139266,-0.491072,0.870802,-0.0234724],[0,-1,-1,0],[9E+09,9E+09,9E+09,9E+09,9E+09,9E+09]],
[[1310.7,118.5,938.01],[0.00139266,-0.491072,0.870802,-0.0234724],[0,-1,-1,0],[9E+09,9E+09,9E+09,9E+09,9E+09,9E+09]],
[[1310.2,119,938.01],[0.00139266,-0.491072,0.870802,-0.0234724],[0,-1,-1,0],[9E+09,9E+09,9E+09,9E+09,9E+09,9E+09]],
[[1309.2,119,938.01],[0.00139266,-0.491072,0.870802,-0.0234724],[0,-1,-1,0],[9E+09,9E+09,9E+09,9E+09,9E+09,9E+09]],
[[1308.7,119.5,938.01],[0.00139266,-0.491072,0.870802,-0.0234724],[0,-1,-1,0],[9E+09,9E+09,9E+09,9E+09,9E+09,9E+09]],
[[1306.2,119.5,938.01],[0.00139266,-0.491072,0.870802,-0.0234724],[0,-1,-1,0],[9E+09,9E+09,9E+09,9E+09,9E+09,9E+09]],
[[1306.2,116.5,938.01],[0.00139266,-0.491072,0.870802,-0.0234724],[0,-1,-1,0],[9E+09,9E+09,9E+09,9E+09,9E+09,9E+09]],
[[1306.7,116,938.01],[0.00139266,-0.491072,0.870802,-0.0234724],[0,-1,-1,0],[9E+09,9E+09,9E+09,9E+09,9E+09,9E+09]],
[[1306.7,115.5,938.01],[0.00139266,-0.491072,0.870802,-0.0234724],[0,-1,-1,0],[9E+09,9E+09,9E+09,9E+09,9E+09,9E+09]],
[[1307.2,115,938.01],[0.00139266,-0.491072,0.870802,-0.0234724],[0,-1,-1,0],[9E+09,9E+09,9E+09,9E+09,9E+09,9E+09]]
];
CONST robtarget myPath2{6} := [
[[1350.7,86.5,938.01],[0.00139266,-0.491072,0.870802,-0.0234724],[0,-1,-1,0],[9E+09,9E+09,9E+09,9E+09,9E+09,9E+09]],
[[1352.2,89,938.01],[0.00139266,-0.491072,0.870802,-0.0234724],[0,-1,-1,0],[9E+09,9E+09,9E+09,9E+09,9E+09,9E+09]],
[[1350.7,95,938.01],[0.00139266,-0.491072,0.870802,-0.0234724],[0,-1,-1,0],[9E+09,9E+09,9E+09,9E+09,9E+09,9E+09]],
[[1348.2,95.5,938.01],[0.00139266,-0.491072,0.870802,-0.0234724],[0,-1,-1,0],[9E+09,9E+09,9E+09,9E+09,9E+09,9E+09]],
[[1345.2,95,938.01],[0.00139266,-0.491072,0.870802,-0.0234724],[0,-1,-1,0],[9E+09,9E+09,9E+09,9E+09,9E+09,9E+09]],
[[1342.2,92.5,938.01],[0.00139266,-0.491072,0.870802,-0.0234724],[0,-1,-1,0],[9E+09,9E+09,9E+09,9E+09,9E+09,9E+09]]
];
CONST robtarget myPath3{146} := [
[[1310.2,72,938.01],[0.00139266,-0.491072,0.870802,-0.0234724],[0,-1,-1,0],[9E+09,9E+09,9E+09,9E+09,9E+09,9E+09]],
[[1317.7,72,938.01],[0.00139266,-0.491072,0.870802,-0.0234724],[0,-1,-1,0],[9E+09,9E+09,9E+09,9E+09,9E+09,9E+09]],
[[1318.2,74.5,938.01],[0.00139266,-0.491072,0.870802,-0.0234724],[0,-1,-1,0],[9E+09,9E+09,9E+09,9E+09,9E+09,9E+09]],
[[1318.7,75,938.01],[0.00139266,-0.491072,0.870802,-0.0234724],[0,-1,-1,0],[9E+09,9E+09,9E+09,9E+09,9E+09,9E+09]],
[[1318.7,75.5,938.01],[0.00139266,-0.491072,0.870802,-0.0234724],[0,-1,-1,0],[9E+09,9E+09,9E+09,9E+09,9E+09,9E+09]],
[[1319.2,76,938.01],[0.00139266,-0.491072,0.870802,-0.0234724],[0,-1,-1,0],[9E+09,9E+09,9E+09,9E+09,9E+09,9E+09]],
[[1319.2,76.5,938.01],[0.00139266,-0.491072,0.870802,-0.0234724],[0,-1,-1,0],[9E+09,9E+09,9E+09,9E+09,9E+09,9E+09]],
[[1319.7,77,938.01],[0.00139266,-0.491072,0.870802,-0.0234724],[0,-1,-1,0],[9E+09,9E+09,9E+09,9E+09,9E+09,9E+09]],
[[1320.2,78.5,938.01],[0.00139266,-0.491072,0.870802,-0.0234724],[0,-1,-1,0],[9E+09,9E+09,9E+09,9E+09,9E+09,9E+09]],
[[1325.7,83,938.01],[0.00139266,-0.491072,0.870802,-0.0234724],[0,-1,-1,0],[9E+09,9E+09,9E+09,9E+09,9E+09,9E+09]],
[[1325.7,83,938.01],[0.00139266,-0.491072,0.870802,-0.0234724],[0,-1,-1,0],[9E+09,9E+09,9E+09,9E+09,9E+09,9E+09]],
[[1326.2,83.5,938.01],[0.00139266,-0.491072,0.870802,-0.0234724],[0,-1,-1,0],[9E+09,9E+09,9E+09,9E+09,9E+09,9E+09]],
[[1326.2,83.5,938.01],[0.00139266,-0.491072,0.870802,-0.0234724],[0,-1,-1,0],[9E+09,9E+09,9E+09,9E+09,9E+09,9E+09]],
[[1330.2,85.5,938.01],[0.00139266,-0.491072,0.870802,-0.0234724],[0,-1,-1,0],[9E+09,9E+09,9E+09,9E+09,9E+09,9E+09]],
[[1330.2,85.5,938.01],[0.00139266,-0.491072,0.870802,-0.0234724],[0,-1,-1,0],[9E+09,9E+09,9E+09,9E+09,9E+09,9E+09]],
[[1330.2,85.5,938.01],[0.00139266,-0.491072,0.870802,-0.0234724],[0,-1,-1,0],[9E+09,9E+09,9E+09,9E+09,9E+09,9E+09]],
[[1330.2,85.5,938.01],[0.00139266,-0.491072,0.870802,-0.0234724],[0,-1,-1,0],[9E+09,9E+09,9E+09,9E+09,9E+09,9E+09]],
[[1331.2,86,938.01],[0.00139266,-0.491072,0.870802,-0.0234724],[0,-1,-1,0],[9E+09,9E+09,9E+09,9E+09,9E+09,9E+09]],
[[1331.2,86,938.01],[0.00139266,-0.491072,0.870802,-0.0234724],[0,-1,-1,0],[9E+09,9E+09,9E+09,9E+09,9E+09,9E+09]],
[[1336.2,88,938.01],[0.00139266,-0.491072,0.870802,-0.0234724],[0,-1,-1,0],[9E+09,9E+09,9E+09,9E+09,9E+09,9E+09]],
[[1336.2,88,938.01],[0.00139266,-0.491072,0.870802,-0.0234724],[0,-1,-1,0],[9E+09,9E+09,9E+09,9E+09,9E+09,9E+09]],
[[1336.2,88,938.01],[0.00139266,-0.491072,0.870802,-0.0234724],[0,-1,-1,0],[9E+09,9E+09,9E+09,9E+09,9E+09,9E+09]],
[[1342.2,89,938.01],[0.00139266,-0.491072,0.870802,-0.0234724],[0,-1,-1,0],[9E+09,9E+09,9E+09,9E+09,9E+09,9E+09]],
[[1342.2,89,938.01],[0.00139266,-0.491072,0.870802,-0.0234724],[0,-1,-1,0],[9E+09,9E+09,9E+09,9E+09,9E+09,9E+09]],
[[1342.2,92.5,938.01],[0.00139266,-0.491072,0.870802,-0.0234724],[0,-1,-1,0],[9E+09,9E+09,9E+09,9E+09,9E+09,9E+09]],
[[1345.2,95,938.01],[0.00139266,-0.491072,0.870802,-0.0234724],[0,-1,-1,0],[9E+09,9E+09,9E+09,9E+09,9E+09,9E+09]],
[[1348.2,95.5,938.01],[0.00139266,-0.491072,0.870802,-0.0234724],[0,-1,-1,0],[9E+09,9E+09,9E+09,9E+09,9E+09,9E+09]],
[[1350.7,95,938.01],[0.00139266,-0.491072,0.870802,-0.0234724],[0,-1,-1,0],[9E+09,9E+09,9E+09,9E+09,9E+09,9E+09]],
[[1352.2,97.5,938.01],[0.00139266,-0.491072,0.870802,-0.0234724],[0,-1,-1,0],[9E+09,9E+09,9E+09,9E+09,9E+09,9E+09]],
[[1352.2,98.5,938.01],[0.00139266,-0.491072,0.870802,-0.0234724],[0,-1,-1,0],[9E+09,9E+09,9E+09,9E+09,9E+09,9E+09]],
[[1352.7,99,938.01],[0.00139266,-0.491072,0.870802,-0.0234724],[0,-1,-1,0],[9E+09,9E+09,9E+09,9E+09,9E+09,9E+09]],
[[1353.2,102.5,938.01],[0.00139266,-0.491072,0.870802,-0.0234724],[0,-1,-1,0],[9E+09,9E+09,9E+09,9E+09,9E+09,9E+09]],
[[1353.2,102.5,938.01],[0.00139266,-0.491072,0.870802,-0.0234724],[0,-1,-1,0],[9E+09,9E+09,9E+09,9E+09,9E+09,9E+09]],
[[1353.2,102.5,938.01],[0.00139266,-0.491072,0.870802,-0.0234724],[0,-1,-1,0],[9E+09,9E+09,9E+09,9E+09,9E+09,9E+09]],
[[1353.2,102.5,938.01],[0.00139266,-0.491072,0.870802,-0.0234724],[0,-1,-1,0],[9E+09,9E+09,9E+09,9E+09,9E+09,9E+09]],
[[1356.2,105,938.01],[0.00139266,-0.491072,0.870802,-0.0234724],[0,-1,-1,0],[9E+09,9E+09,9E+09,9E+09,9E+09,9E+09]],
[[1356.7,108,938.01],[0.00139266,-0.491072,0.870802,-0.0234724],[0,-1,-1,0],[9E+09,9E+09,9E+09,9E+09,9E+09,9E+09]],
[[1352.7,111,938.01],[0.00139266,-0.491072,0.870802,-0.0234724],[0,-1,-1,0],[9E+09,9E+09,9E+09,9E+09,9E+09,9E+09]],
[[1352.7,111,938.01],[0.00139266,-0.491072,0.870802,-0.0234724],[0,-1,-1,0],[9E+09,9E+09,9E+09,9E+09,9E+09,9E+09]],
[[1352.7,111,938.01],[0.00139266,-0.491072,0.870802,-0.0234724],[0,-1,-1,0],[9E+09,9E+09,9E+09,9E+09,9E+09,9E+09]],
[[1349.2,112,938.01],[0.00139266,-0.491072,0.870802,-0.0234724],[0,-1,-1,0],[9E+09,9E+09,9E+09,9E+09,9E+09,9E+09]],
[[1348.7,112.5,938.01],[0.00139266,-0.491072,0.870802,-0.0234724],[0,-1,-1,0],[9E+09,9E+09,9E+09,9E+09,9E+09,9E+09]],
[[1347.2,112.5,938.01],[0.00139266,-0.491072,0.870802,-0.0234724],[0,-1,-1,0],[9E+09,9E+09,9E+09,9E+09,9E+09,9E+09]],
[[1346.7,113,938.01],[0.00139266,-0.491072,0.870802,-0.0234724],[0,-1,-1,0],[9E+09,9E+09,9E+09,9E+09,9E+09,9E+09]],
[[1343.7,113.5,938.01],[0.00139266,-0.491072,0.870802,-0.0234724],[0,-1,-1,0],[9E+09,9E+09,9E+09,9E+09,9E+09,9E+09]],
[[1343.7,113.5,938.01],[0.00139266,-0.491072,0.870802,-0.0234724],[0,-1,-1,0],[9E+09,9E+09,9E+09,9E+09,9E+09,9E+09]],
[[1342.7,111,938.01],[0.00139266,-0.491072,0.870802,-0.0234724],[0,-1,-1,0],[9E+09,9E+09,9E+09,9E+09,9E+09,9E+09]],
[[1342.7,107.5,938.01],[0.00139266,-0.491072,0.870802,-0.0234724],[0,-1,-1,0],[9E+09,9E+09,9E+09,9E+09,9E+09,9E+09]],
[[1342.2,107,938.01],[0.00139266,-0.491072,0.870802,-0.0234724],[0,-1,-1,0],[9E+09,9E+09,9E+09,9E+09,9E+09,9E+09]],
[[1341.7,104.5,938.01],[0.00139266,-0.491072,0.870802,-0.0234724],[0,-1,-1,0],[9E+09,9E+09,9E+09,9E+09,9E+09,9E+09]],
[[1341.7,104.5,938.01],[0.00139266,-0.491072,0.870802,-0.0234724],[0,-1,-1,0],[9E+09,9E+09,9E+09,9E+09,9E+09,9E+09]],
[[1340.2,101,938.01],[0.00139266,-0.491072,0.870802,-0.0234724],[0,-1,-1,0],[9E+09,9E+09,9E+09,9E+09,9E+09,9E+09]],
[[1340.2,101,938.01],[0.00139266,-0.491072,0.870802,-0.0234724],[0,-1,-1,0],[9E+09,9E+09,9E+09,9E+09,9E+09,9E+09]],
[[1341.7,104.5,938.01],[0.00139266,-0.491072,0.870802,-0.0234724],[0,-1,-1,0],[9E+09,9E+09,9E+09,9E+09,9E+09,9E+09]],
[[1342.2,107,938.01],[0.00139266,-0.491072,0.870802,-0.0234724],[0,-1,-1,0],[9E+09,9E+09,9E+09,9E+09,9E+09,9E+09]],
[[1342.7,107.5,938.01],[0.00139266,-0.491072,0.870802,-0.0234724],[0,-1,-1,0],[9E+09,9E+09,9E+09,9E+09,9E+09,9E+09]],
[[1342.7,111,938.01],[0.00139266,-0.491072,0.870802,-0.0234724],[0,-1,-1,0],[9E+09,9E+09,9E+09,9E+09,9E+09,9E+09]],
[[1343.7,113.5,938.01],[0.00139266,-0.491072,0.870802,-0.0234724],[0,-1,-1,0],[9E+09,9E+09,9E+09,9E+09,9E+09,9E+09]],
[[1343.7,113.5,938.01],[0.00139266,-0.491072,0.870802,-0.0234724],[0,-1,-1,0],[9E+09,9E+09,9E+09,9E+09,9E+09,9E+09]],
[[1345.2,119,938.01],[0.00139266,-0.491072,0.870802,-0.0234724],[0,-1,-1,0],[9E+09,9E+09,9E+09,9E+09,9E+09,9E+09]],
[[1345.2,119,938.01],[0.00139266,-0.491072,0.870802,-0.0234724],[0,-1,-1,0],[9E+09,9E+09,9E+09,9E+09,9E+09,9E+09]],
[[1343.2,120.5,938.01],[0.00139266,-0.491072,0.870802,-0.0234724],[0,-1,-1,0],[9E+09,9E+09,9E+09,9E+09,9E+09,9E+09]],
[[1342.7,121,938.01],[0.00139266,-0.491072,0.870802,-0.0234724],[0,-1,-1,0],[9E+09,9E+09,9E+09,9E+09,9E+09,9E+09]],
[[1341.2,121,938.01],[0.00139266,-0.491072,0.870802,-0.0234724],[0,-1,-1,0],[9E+09,9E+09,9E+09,9E+09,9E+09,9E+09]],
[[1340.7,121.5,938.01],[0.00139266,-0.491072,0.870802,-0.0234724],[0,-1,-1,0],[9E+09,9E+09,9E+09,9E+09,9E+09,9E+09]],
[[1325.2,120,938.01],[0.00139266,-0.491072,0.870802,-0.0234724],[0,-1,-1,0],[9E+09,9E+09,9E+09,9E+09,9E+09,9E+09]],
[[1325.2,120,938.01],[0.00139266,-0.491072,0.870802,-0.0234724],[0,-1,-1,0],[9E+09,9E+09,9E+09,9E+09,9E+09,9E+09]],
[[1325.2,120,938.01],[0.00139266,-0.491072,0.870802,-0.0234724],[0,-1,-1,0],[9E+09,9E+09,9E+09,9E+09,9E+09,9E+09]],
[[1322.7,118,938.01],[0.00139266,-0.491072,0.870802,-0.0234724],[0,-1,-1,0],[9E+09,9E+09,9E+09,9E+09,9E+09,9E+09]],
[[1320.2,114,938.01],[0.00139266,-0.491072,0.870802,-0.0234724],[0,-1,-1,0],[9E+09,9E+09,9E+09,9E+09,9E+09,9E+09]],
[[1320.2,114,938.01],[0.00139266,-0.491072,0.870802,-0.0234724],[0,-1,-1,0],[9E+09,9E+09,9E+09,9E+09,9E+09,9E+09]],
[[1320.2,114,938.01],[0.00139266,-0.491072,0.870802,-0.0234724],[0,-1,-1,0],[9E+09,9E+09,9E+09,9E+09,9E+09,9E+09]],
[[1314.2,114,938.01],[0.00139266,-0.491072,0.870802,-0.0234724],[0,-1,-1,0],[9E+09,9E+09,9E+09,9E+09,9E+09,9E+09]],
[[1313.7,113.5,938.01],[0.00139266,-0.491072,0.870802,-0.0234724],[0,-1,-1,0],[9E+09,9E+09,9E+09,9E+09,9E+09,9E+09]],
[[1312.2,113.5,938.01],[0.00139266,-0.491072,0.870802,-0.0234724],[0,-1,-1,0],[9E+09,9E+09,9E+09,9E+09,9E+09,9E+09]],
[[1311.7,113,938.01],[0.00139266,-0.491072,0.870802,-0.0234724],[0,-1,-1,0],[9E+09,9E+09,9E+09,9E+09,9E+09,9E+09]],
[[1308.7,112,938.01],[0.00139266,-0.491072,0.870802,-0.0234724],[0,-1,-1,0],[9E+09,9E+09,9E+09,9E+09,9E+09,9E+09]],
[[1308.7,112,938.01],[0.00139266,-0.491072,0.870802,-0.0234724],[0,-1,-1,0],[9E+09,9E+09,9E+09,9E+09,9E+09,9E+09]],
[[1308.7,112,938.01],[0.00139266,-0.491072,0.870802,-0.0234724],[0,-1,-1,0],[9E+09,9E+09,9E+09,9E+09,9E+09,9E+09]],
[[1309.2,109.5,938.01],[0.00139266,-0.491072,0.870802,-0.0234724],[0,-1,-1,0],[9E+09,9E+09,9E+09,9E+09,9E+09,9E+09]],
[[1308.7,99.5,938.01],[0.00139266,-0.491072,0.870802,-0.0234724],[0,-1,-1,0],[9E+09,9E+09,9E+09,9E+09,9E+09,9E+09]],
[[1308.7,99.5,938.01],[0.00139266,-0.491072,0.870802,-0.0234724],[0,-1,-1,0],[9E+09,9E+09,9E+09,9E+09,9E+09,9E+09]],
[[1308.2,98.5,938.01],[0.00139266,-0.491072,0.870802,-0.0234724],[0,-1,-1,0],[9E+09,9E+09,9E+09,9E+09,9E+09,9E+09]],
[[1308.2,98.5,938.01],[0.00139266,-0.491072,0.870802,-0.0234724],[0,-1,-1,0],[9E+09,9E+09,9E+09,9E+09,9E+09,9E+09]],
[[1308.2,98,938.01],[0.00139266,-0.491072,0.870802,-0.0234724],[0,-1,-1,0],[9E+09,9E+09,9E+09,9E+09,9E+09,9E+09]],
[[1306.2,95.5,938.01],[0.00139266,-0.491072,0.870802,-0.0234724],[0,-1,-1,0],[9E+09,9E+09,9E+09,9E+09,9E+09,9E+09]],
[[1306.2,95.5,938.01],[0.00139266,-0.491072,0.870802,-0.0234724],[0,-1,-1,0],[9E+09,9E+09,9E+09,9E+09,9E+09,9E+09]],
[[1306.2,95.5,938.01],[0.00139266,-0.491072,0.870802,-0.0234724],[0,-1,-1,0],[9E+09,9E+09,9E+09,9E+09,9E+09,9E+09]],
[[1306.2,95.5,938.01],[0.00139266,-0.491072,0.870802,-0.0234724],[0,-1,-1,0],[9E+09,9E+09,9E+09,9E+09,9E+09,9E+09]],
[[1308.2,98,938.01],[0.00139266,-0.491072,0.870802,-0.0234724],[0,-1,-1,0],[9E+09,9E+09,9E+09,9E+09,9E+09,9E+09]],
[[1308.2,98.5,938.01],[0.00139266,-0.491072,0.870802,-0.0234724],[0,-1,-1,0],[9E+09,9E+09,9E+09,9E+09,9E+09,9E+09]],
[[1308.7,99.5,938.01],[0.00139266,-0.491072,0.870802,-0.0234724],[0,-1,-1,0],[9E+09,9E+09,9E+09,9E+09,9E+09,9E+09]],
[[1308.7,99.5,938.01],[0.00139266,-0.491072,0.870802,-0.0234724],[0,-1,-1,0],[9E+09,9E+09,9E+09,9E+09,9E+09,9E+09]],
[[1309.2,109.5,938.01],[0.00139266,-0.491072,0.870802,-0.0234724],[0,-1,-1,0],[9E+09,9E+09,9E+09,9E+09,9E+09,9E+09]],
[[1307.2,115,938.01],[0.00139266,-0.491072,0.870802,-0.0234724],[0,-1,-1,0],[9E+09,9E+09,9E+09,9E+09,9E+09,9E+09]],
[[1306.7,115.5,938.01],[0.00139266,-0.491072,0.870802,-0.0234724],[0,-1,-1,0],[9E+09,9E+09,9E+09,9E+09,9E+09,9E+09]],
[[1306.7,116,938.01],[0.00139266,-0.491072,0.870802,-0.0234724],[0,-1,-1,0],[9E+09,9E+09,9E+09,9E+09,9E+09,9E+09]],
[[1306.2,116.5,938.01],[0.00139266,-0.491072,0.870802,-0.0234724],[0,-1,-1,0],[9E+09,9E+09,9E+09,9E+09,9E+09,9E+09]],
[[1306.2,119.5,938.01],[0.00139266,-0.491072,0.870802,-0.0234724],[0,-1,-1,0],[9E+09,9E+09,9E+09,9E+09,9E+09,9E+09]],
[[1303.2,120.5,938.01],[0.00139266,-0.491072,0.870802,-0.0234724],[0,-1,-1,0],[9E+09,9E+09,9E+09,9E+09,9E+09,9E+09]],
[[1302.7,121,938.01],[0.00139266,-0.491072,0.870802,-0.0234724],[0,-1,-1,0],[9E+09,9E+09,9E+09,9E+09,9E+09,9E+09]],
[[1301.7,121,938.01],[0.00139266,-0.491072,0.870802,-0.0234724],[0,-1,-1,0],[9E+09,9E+09,9E+09,9E+09,9E+09,9E+09]],
[[1301.2,121.5,938.01],[0.00139266,-0.491072,0.870802,-0.0234724],[0,-1,-1,0],[9E+09,9E+09,9E+09,9E+09,9E+09,9E+09]],
[[1292.2,121.5,938.01],[0.00139266,-0.491072,0.870802,-0.0234724],[0,-1,-1,0],[9E+09,9E+09,9E+09,9E+09,9E+09,9E+09]],
[[1290.2,120.5,938.01],[0.00139266,-0.491072,0.870802,-0.0234724],[0,-1,-1,0],[9E+09,9E+09,9E+09,9E+09,9E+09,9E+09]],
[[1288.2,119.5,938.01],[0.00139266,-0.491072,0.870802,-0.0234724],[0,-1,-1,0],[9E+09,9E+09,9E+09,9E+09,9E+09,9E+09]],
[[1287.2,119,938.01],[0.00139266,-0.491072,0.870802,-0.0234724],[0,-1,-1,0],[9E+09,9E+09,9E+09,9E+09,9E+09,9E+09]],
[[1285.7,118,938.01],[0.00139266,-0.491072,0.870802,-0.0234724],[0,-1,-1,0],[9E+09,9E+09,9E+09,9E+09,9E+09,9E+09]],
[[1285.7,117.5,938.01],[0.00139266,-0.491072,0.870802,-0.0234724],[0,-1,-1,0],[9E+09,9E+09,9E+09,9E+09,9E+09,9E+09]],
[[1280.7,111,938.01],[0.00139266,-0.491072,0.870802,-0.0234724],[0,-1,-1,0],[9E+09,9E+09,9E+09,9E+09,9E+09,9E+09]],
[[1280.7,111,938.01],[0.00139266,-0.491072,0.870802,-0.0234724],[0,-1,-1,0],[9E+09,9E+09,9E+09,9E+09,9E+09,9E+09]],
[[1280.2,110.5,938.01],[0.00139266,-0.491072,0.870802,-0.0234724],[0,-1,-1,0],[9E+09,9E+09,9E+09,9E+09,9E+09,9E+09]],
[[1280.2,110.5,938.01],[0.00139266,-0.491072,0.870802,-0.0234724],[0,-1,-1,0],[9E+09,9E+09,9E+09,9E+09,9E+09,9E+09]],
[[1279.7,109.5,938.01],[0.00139266,-0.491072,0.870802,-0.0234724],[0,-1,-1,0],[9E+09,9E+09,9E+09,9E+09,9E+09,9E+09]],
[[1279.7,109.5,938.01],[0.00139266,-0.491072,0.870802,-0.0234724],[0,-1,-1,0],[9E+09,9E+09,9E+09,9E+09,9E+09,9E+09]],
[[1279.7,109,938.01],[0.00139266,-0.491072,0.870802,-0.0234724],[0,-1,-1,0],[9E+09,9E+09,9E+09,9E+09,9E+09,9E+09]],
[[1279.2,108,938.01],[0.00139266,-0.491072,0.870802,-0.0234724],[0,-1,-1,0],[9E+09,9E+09,9E+09,9E+09,9E+09,9E+09]],
[[1278.7,106,938.01],[0.00139266,-0.491072,0.870802,-0.0234724],[0,-1,-1,0],[9E+09,9E+09,9E+09,9E+09,9E+09,9E+09]],
[[1278.2,94.5,938.01],[0.00139266,-0.491072,0.870802,-0.0234724],[0,-1,-1,0],[9E+09,9E+09,9E+09,9E+09,9E+09,9E+09]],
[[1278.7,94,938.01],[0.00139266,-0.491072,0.870802,-0.0234724],[0,-1,-1,0],[9E+09,9E+09,9E+09,9E+09,9E+09,9E+09]],
[[1278.7,93,938.01],[0.00139266,-0.491072,0.870802,-0.0234724],[0,-1,-1,0],[9E+09,9E+09,9E+09,9E+09,9E+09,9E+09]],
[[1279.2,92.5,938.01],[0.00139266,-0.491072,0.870802,-0.0234724],[0,-1,-1,0],[9E+09,9E+09,9E+09,9E+09,9E+09,9E+09]],
[[1279.7,90,938.01],[0.00139266,-0.491072,0.870802,-0.0234724],[0,-1,-1,0],[9E+09,9E+09,9E+09,9E+09,9E+09,9E+09]],
[[1279.7,90,938.01],[0.00139266,-0.491072,0.870802,-0.0234724],[0,-1,-1,0],[9E+09,9E+09,9E+09,9E+09,9E+09,9E+09]],
[[1279.7,90,938.01],[0.00139266,-0.491072,0.870802,-0.0234724],[0,-1,-1,0],[9E+09,9E+09,9E+09,9E+09,9E+09,9E+09]],
[[1281.7,87,938.01],[0.00139266,-0.491072,0.870802,-0.0234724],[0,-1,-1,0],[9E+09,9E+09,9E+09,9E+09,9E+09,9E+09]],
[[1281.7,86.5,938.01],[0.00139266,-0.491072,0.870802,-0.0234724],[0,-1,-1,0],[9E+09,9E+09,9E+09,9E+09,9E+09,9E+09]],
[[1282.2,86,938.01],[0.00139266,-0.491072,0.870802,-0.0234724],[0,-1,-1,0],[9E+09,9E+09,9E+09,9E+09,9E+09,9E+09]],
[[1282.2,85.5,938.01],[0.00139266,-0.491072,0.870802,-0.0234724],[0,-1,-1,0],[9E+09,9E+09,9E+09,9E+09,9E+09,9E+09]],
[[1286.7,80.5,938.01],[0.00139266,-0.491072,0.870802,-0.0234724],[0,-1,-1,0],[9E+09,9E+09,9E+09,9E+09,9E+09,9E+09]],
[[1286.7,80.5,938.01],[0.00139266,-0.491072,0.870802,-0.0234724],[0,-1,-1,0],[9E+09,9E+09,9E+09,9E+09,9E+09,9E+09]],
[[1292.2,77.5,938.01],[0.00139266,-0.491072,0.870802,-0.0234724],[0,-1,-1,0],[9E+09,9E+09,9E+09,9E+09,9E+09,9E+09]],
[[1292.2,77.5,938.01],[0.00139266,-0.491072,0.870802,-0.0234724],[0,-1,-1,0],[9E+09,9E+09,9E+09,9E+09,9E+09,9E+09]],
[[1292.2,77.5,938.01],[0.00139266,-0.491072,0.870802,-0.0234724],[0,-1,-1,0],[9E+09,9E+09,9E+09,9E+09,9E+09,9E+09]],
[[1292.7,77.5,938.01],[0.00139266,-0.491072,0.870802,-0.0234724],[0,-1,-1,0],[9E+09,9E+09,9E+09,9E+09,9E+09,9E+09]],
[[1293.2,77,938.01],[0.00139266,-0.491072,0.870802,-0.0234724],[0,-1,-1,0],[9E+09,9E+09,9E+09,9E+09,9E+09,9E+09]],
[[1294.2,76.5,938.01],[0.00139266,-0.491072,0.870802,-0.0234724],[0,-1,-1,0],[9E+09,9E+09,9E+09,9E+09,9E+09,9E+09]],
[[1295.2,76.5,938.01],[0.00139266,-0.491072,0.870802,-0.0234724],[0,-1,-1,0],[9E+09,9E+09,9E+09,9E+09,9E+09,9E+09]],
[[1295.7,76,938.01],[0.00139266,-0.491072,0.870802,-0.0234724],[0,-1,-1,0],[9E+09,9E+09,9E+09,9E+09,9E+09,9E+09]],
[[1295.7,76,938.01],[0.00139266,-0.491072,0.870802,-0.0234724],[0,-1,-1,0],[9E+09,9E+09,9E+09,9E+09,9E+09,9E+09]],
[[1295.7,76,938.01],[0.00139266,-0.491072,0.870802,-0.0234724],[0,-1,-1,0],[9E+09,9E+09,9E+09,9E+09,9E+09,9E+09]],
[[1295.7,76,938.01],[0.00139266,-0.491072,0.870802,-0.0234724],[0,-1,-1,0],[9E+09,9E+09,9E+09,9E+09,9E+09,9E+09]],
[[1299.2,75,938.01],[0.00139266,-0.491072,0.870802,-0.0234724],[0,-1,-1,0],[9E+09,9E+09,9E+09,9E+09,9E+09,9E+09]],
[[1299.7,74.5,938.01],[0.00139266,-0.491072,0.870802,-0.0234724],[0,-1,-1,0],[9E+09,9E+09,9E+09,9E+09,9E+09,9E+09]],
[[1301.2,74.5,938.01],[0.00139266,-0.491072,0.870802,-0.0234724],[0,-1,-1,0],[9E+09,9E+09,9E+09,9E+09,9E+09,9E+09]],
[[1301.7,74,938.01],[0.00139266,-0.491072,0.870802,-0.0234724],[0,-1,-1,0],[9E+09,9E+09,9E+09,9E+09,9E+09,9E+09]]
];
CONST robtarget myPath4{43} := [
[[1323.7,70,938.01],[0.00139266,-0.491072,0.870802,-0.0234724],[0,-1,-1,0],[9E+09,9E+09,9E+09,9E+09,9E+09,9E+09]],
[[1323.7,70,938.01],[0.00139266,-0.491072,0.870802,-0.0234724],[0,-1,-1,0],[9E+09,9E+09,9E+09,9E+09,9E+09,9E+09]],
[[1329.7,75.5,938.01],[0.00139266,-0.491072,0.870802,-0.0234724],[0,-1,-1,0],[9E+09,9E+09,9E+09,9E+09,9E+09,9E+09]],
[[1329.7,75.5,938.01],[0.00139266,-0.491072,0.870802,-0.0234724],[0,-1,-1,0],[9E+09,9E+09,9E+09,9E+09,9E+09,9E+09]],
[[1329.7,75.5,938.01],[0.00139266,-0.491072,0.870802,-0.0234724],[0,-1,-1,0],[9E+09,9E+09,9E+09,9E+09,9E+09,9E+09]],
[[1330.7,76,938.01],[0.00139266,-0.491072,0.870802,-0.0234724],[0,-1,-1,0],[9E+09,9E+09,9E+09,9E+09,9E+09,9E+09]],
[[1330.7,76,938.01],[0.00139266,-0.491072,0.870802,-0.0234724],[0,-1,-1,0],[9E+09,9E+09,9E+09,9E+09,9E+09,9E+09]],
[[1332.7,77,938.01],[0.00139266,-0.491072,0.870802,-0.0234724],[0,-1,-1,0],[9E+09,9E+09,9E+09,9E+09,9E+09,9E+09]],
[[1333.7,77.5,938.01],[0.00139266,-0.491072,0.870802,-0.0234724],[0,-1,-1,0],[9E+09,9E+09,9E+09,9E+09,9E+09,9E+09]],
[[1336.7,78.5,938.01],[0.00139266,-0.491072,0.870802,-0.0234724],[0,-1,-1,0],[9E+09,9E+09,9E+09,9E+09,9E+09,9E+09]],
[[1338.7,79.5,938.01],[0.00139266,-0.491072,0.870802,-0.0234724],[0,-1,-1,0],[9E+09,9E+09,9E+09,9E+09,9E+09,9E+09]],
[[1338.7,79.5,938.01],[0.00139266,-0.491072,0.870802,-0.0234724],[0,-1,-1,0],[9E+09,9E+09,9E+09,9E+09,9E+09,9E+09]],
[[1338.7,79.5,938.01],[0.00139266,-0.491072,0.870802,-0.0234724],[0,-1,-1,0],[9E+09,9E+09,9E+09,9E+09,9E+09,9E+09]],
[[1353.7,81,938.01],[0.00139266,-0.491072,0.870802,-0.0234724],[0,-1,-1,0],[9E+09,9E+09,9E+09,9E+09,9E+09,9E+09]],
[[1353.7,81,938.01],[0.00139266,-0.491072,0.870802,-0.0234724],[0,-1,-1,0],[9E+09,9E+09,9E+09,9E+09,9E+09,9E+09]],
[[1350.7,86.5,938.01],[0.00139266,-0.491072,0.870802,-0.0234724],[0,-1,-1,0],[9E+09,9E+09,9E+09,9E+09,9E+09,9E+09]],
[[1350.7,86.5,938.01],[0.00139266,-0.491072,0.870802,-0.0234724],[0,-1,-1,0],[9E+09,9E+09,9E+09,9E+09,9E+09,9E+09]],
[[1345.2,86,938.01],[0.00139266,-0.491072,0.870802,-0.0234724],[0,-1,-1,0],[9E+09,9E+09,9E+09,9E+09,9E+09,9E+09]],
[[1342.2,89,938.01],[0.00139266,-0.491072,0.870802,-0.0234724],[0,-1,-1,0],[9E+09,9E+09,9E+09,9E+09,9E+09,9E+09]],
[[1342.2,89,938.01],[0.00139266,-0.491072,0.870802,-0.0234724],[0,-1,-1,0],[9E+09,9E+09,9E+09,9E+09,9E+09,9E+09]],
[[1342.2,89,938.01],[0.00139266,-0.491072,0.870802,-0.0234724],[0,-1,-1,0],[9E+09,9E+09,9E+09,9E+09,9E+09,9E+09]],
[[1342.2,89,938.01],[0.00139266,-0.491072,0.870802,-0.0234724],[0,-1,-1,0],[9E+09,9E+09,9E+09,9E+09,9E+09,9E+09]],
[[1342.2,89,938.01],[0.00139266,-0.491072,0.870802,-0.0234724],[0,-1,-1,0],[9E+09,9E+09,9E+09,9E+09,9E+09,9E+09]],
[[1336.2,88,938.01],[0.00139266,-0.491072,0.870802,-0.0234724],[0,-1,-1,0],[9E+09,9E+09,9E+09,9E+09,9E+09,9E+09]],
[[1336.2,88,938.01],[0.00139266,-0.491072,0.870802,-0.0234724],[0,-1,-1,0],[9E+09,9E+09,9E+09,9E+09,9E+09,9E+09]],
[[1336.2,88,938.01],[0.00139266,-0.491072,0.870802,-0.0234724],[0,-1,-1,0],[9E+09,9E+09,9E+09,9E+09,9E+09,9E+09]],
[[1331.2,86,938.01],[0.00139266,-0.491072,0.870802,-0.0234724],[0,-1,-1,0],[9E+09,9E+09,9E+09,9E+09,9E+09,9E+09]],
[[1331.2,86,938.01],[0.00139266,-0.491072,0.870802,-0.0234724],[0,-1,-1,0],[9E+09,9E+09,9E+09,9E+09,9E+09,9E+09]],
[[1330.2,85.5,938.01],[0.00139266,-0.491072,0.870802,-0.0234724],[0,-1,-1,0],[9E+09,9E+09,9E+09,9E+09,9E+09,9E+09]],
[[1330.2,85.5,938.01],[0.00139266,-0.491072,0.870802,-0.0234724],[0,-1,-1,0],[9E+09,9E+09,9E+09,9E+09,9E+09,9E+09]],
[[1330.2,85.5,938.01],[0.00139266,-0.491072,0.870802,-0.0234724],[0,-1,-1,0],[9E+09,9E+09,9E+09,9E+09,9E+09,9E+09]],
[[1330.2,85.5,938.01],[0.00139266,-0.491072,0.870802,-0.0234724],[0,-1,-1,0],[9E+09,9E+09,9E+09,9E+09,9E+09,9E+09]],
[[1325.7,83,938.01],[0.00139266,-0.491072,0.870802,-0.0234724],[0,-1,-1,0],[9E+09,9E+09,9E+09,9E+09,9E+09,9E+09]],
[[1325.7,83,938.01],[0.00139266,-0.491072,0.870802,-0.0234724],[0,-1,-1,0],[9E+09,9E+09,9E+09,9E+09,9E+09,9E+09]],
[[1324.2,82,938.01],[0.00139266,-0.491072,0.870802,-0.0234724],[0,-1,-1,0],[9E+09,9E+09,9E+09,9E+09,9E+09,9E+09]],
[[1322.7,81,938.01],[0.00139266,-0.491072,0.870802,-0.0234724],[0,-1,-1,0],[9E+09,9E+09,9E+09,9E+09,9E+09,9E+09]],
[[1320.2,78.5,938.01],[0.00139266,-0.491072,0.870802,-0.0234724],[0,-1,-1,0],[9E+09,9E+09,9E+09,9E+09,9E+09,9E+09]],
[[1319.7,77,938.01],[0.00139266,-0.491072,0.870802,-0.0234724],[0,-1,-1,0],[9E+09,9E+09,9E+09,9E+09,9E+09,9E+09]],
[[1319.2,76.5,938.01],[0.00139266,-0.491072,0.870802,-0.0234724],[0,-1,-1,0],[9E+09,9E+09,9E+09,9E+09,9E+09,9E+09]],
[[1319.2,76,938.01],[0.00139266,-0.491072,0.870802,-0.0234724],[0,-1,-1,0],[9E+09,9E+09,9E+09,9E+09,9E+09,9E+09]],
[[1318.7,75.5,938.01],[0.00139266,-0.491072,0.870802,-0.0234724],[0,-1,-1,0],[9E+09,9E+09,9E+09,9E+09,9E+09,9E+09]],
[[1318.7,75,938.01],[0.00139266,-0.491072,0.870802,-0.0234724],[0,-1,-1,0],[9E+09,9E+09,9E+09,9E+09,9E+09,9E+09]],
[[1318.2,74.5,938.01],[0.00139266,-0.491072,0.870802,-0.0234724],[0,-1,-1,0],[9E+09,9E+09,9E+09,9E+09,9E+09,9E+09]]
];
CONST robtarget myPath5{38} := [
[[1281.2,63,938.01],[0.00139266,-0.491072,0.870802,-0.0234724],[0,-1,-1,0],[9E+09,9E+09,9E+09,9E+09,9E+09,9E+09]],
[[1281.2,68.5,938.01],[0.00139266,-0.491072,0.870802,-0.0234724],[0,-1,-1,0],[9E+09,9E+09,9E+09,9E+09,9E+09,9E+09]],
[[1280.7,75,938.01],[0.00139266,-0.491072,0.870802,-0.0234724],[0,-1,-1,0],[9E+09,9E+09,9E+09,9E+09,9E+09,9E+09]],
[[1286.7,80.5,938.01],[0.00139266,-0.491072,0.870802,-0.0234724],[0,-1,-1,0],[9E+09,9E+09,9E+09,9E+09,9E+09,9E+09]],
[[1286.7,80.5,938.01],[0.00139266,-0.491072,0.870802,-0.0234724],[0,-1,-1,0],[9E+09,9E+09,9E+09,9E+09,9E+09,9E+09]],
[[1286.7,80.5,938.01],[0.00139266,-0.491072,0.870802,-0.0234724],[0,-1,-1,0],[9E+09,9E+09,9E+09,9E+09,9E+09,9E+09]],
[[1284.2,83,938.01],[0.00139266,-0.491072,0.870802,-0.0234724],[0,-1,-1,0],[9E+09,9E+09,9E+09,9E+09,9E+09,9E+09]],
[[1284.2,83.5,938.01],[0.00139266,-0.491072,0.870802,-0.0234724],[0,-1,-1,0],[9E+09,9E+09,9E+09,9E+09,9E+09,9E+09]],
[[1282.2,85.5,938.01],[0.00139266,-0.491072,0.870802,-0.0234724],[0,-1,-1,0],[9E+09,9E+09,9E+09,9E+09,9E+09,9E+09]],
[[1282.2,86,938.01],[0.00139266,-0.491072,0.870802,-0.0234724],[0,-1,-1,0],[9E+09,9E+09,9E+09,9E+09,9E+09,9E+09]],
[[1281.7,86.5,938.01],[0.00139266,-0.491072,0.870802,-0.0234724],[0,-1,-1,0],[9E+09,9E+09,9E+09,9E+09,9E+09,9E+09]],
[[1281.7,87,938.01],[0.00139266,-0.491072,0.870802,-0.0234724],[0,-1,-1,0],[9E+09,9E+09,9E+09,9E+09,9E+09,9E+09]],
[[1279.7,90,938.01],[0.00139266,-0.491072,0.870802,-0.0234724],[0,-1,-1,0],[9E+09,9E+09,9E+09,9E+09,9E+09,9E+09]],
[[1279.7,90,938.01],[0.00139266,-0.491072,0.870802,-0.0234724],[0,-1,-1,0],[9E+09,9E+09,9E+09,9E+09,9E+09,9E+09]],
[[1279.7,90,938.01],[0.00139266,-0.491072,0.870802,-0.0234724],[0,-1,-1,0],[9E+09,9E+09,9E+09,9E+09,9E+09,9E+09]],
[[1275.7,90,938.01],[0.00139266,-0.491072,0.870802,-0.0234724],[0,-1,-1,0],[9E+09,9E+09,9E+09,9E+09,9E+09,9E+09]],
[[1275.2,89.5,938.01],[0.00139266,-0.491072,0.870802,-0.0234724],[0,-1,-1,0],[9E+09,9E+09,9E+09,9E+09,9E+09,9E+09]],
[[1270.7,88.5,938.01],[0.00139266,-0.491072,0.870802,-0.0234724],[0,-1,-1,0],[9E+09,9E+09,9E+09,9E+09,9E+09,9E+09]],
[[1270.2,88,938.01],[0.00139266,-0.491072,0.870802,-0.0234724],[0,-1,-1,0],[9E+09,9E+09,9E+09,9E+09,9E+09,9E+09]],
[[1270.2,88,938.01],[0.00139266,-0.491072,0.870802,-0.0234724],[0,-1,-1,0],[9E+09,9E+09,9E+09,9E+09,9E+09,9E+09]],
[[1266.7,85,938.01],[0.00139266,-0.491072,0.870802,-0.0234724],[0,-1,-1,0],[9E+09,9E+09,9E+09,9E+09,9E+09,9E+09]],
[[1266.2,84,938.01],[0.00139266,-0.491072,0.870802,-0.0234724],[0,-1,-1,0],[9E+09,9E+09,9E+09,9E+09,9E+09,9E+09]],
[[1265.7,83.5,938.01],[0.00139266,-0.491072,0.870802,-0.0234724],[0,-1,-1,0],[9E+09,9E+09,9E+09,9E+09,9E+09,9E+09]],
[[1265.2,76.5,938.01],[0.00139266,-0.491072,0.870802,-0.0234724],[0,-1,-1,0],[9E+09,9E+09,9E+09,9E+09,9E+09,9E+09]],
[[1266.2,74,938.01],[0.00139266,-0.491072,0.870802,-0.0234724],[0,-1,-1,0],[9E+09,9E+09,9E+09,9E+09,9E+09,9E+09]],
[[1266.2,74,938.01],[0.00139266,-0.491072,0.870802,-0.0234724],[0,-1,-1,0],[9E+09,9E+09,9E+09,9E+09,9E+09,9E+09]],
[[1266.2,74,938.01],[0.00139266,-0.491072,0.870802,-0.0234724],[0,-1,-1,0],[9E+09,9E+09,9E+09,9E+09,9E+09,9E+09]],
[[1266.2,74,938.01],[0.00139266,-0.491072,0.870802,-0.0234724],[0,-1,-1,0],[9E+09,9E+09,9E+09,9E+09,9E+09,9E+09]],
[[1273.2,66.5,938.01],[0.00139266,-0.491072,0.870802,-0.0234724],[0,-1,-1,0],[9E+09,9E+09,9E+09,9E+09,9E+09,9E+09]],
[[1273.2,66,938.01],[0.00139266,-0.491072,0.870802,-0.0234724],[0,-1,-1,0],[9E+09,9E+09,9E+09,9E+09,9E+09,9E+09]],
[[1273.7,66,938.01],[0.00139266,-0.491072,0.870802,-0.0234724],[0,-1,-1,0],[9E+09,9E+09,9E+09,9E+09,9E+09,9E+09]],
[[1274.2,66,938.01],[0.00139266,-0.491072,0.870802,-0.0234724],[0,-1,-1,0],[9E+09,9E+09,9E+09,9E+09,9E+09,9E+09]],
[[1275.7,65,938.01],[0.00139266,-0.491072,0.870802,-0.0234724],[0,-1,-1,0],[9E+09,9E+09,9E+09,9E+09,9E+09,9E+09]],
[[1275.7,65,938.01],[0.00139266,-0.491072,0.870802,-0.0234724],[0,-1,-1,0],[9E+09,9E+09,9E+09,9E+09,9E+09,9E+09]],
[[1276.2,64.5,938.01],[0.00139266,-0.491072,0.870802,-0.0234724],[0,-1,-1,0],[9E+09,9E+09,9E+09,9E+09,9E+09,9E+09]],
[[1276.7,64.5,938.01],[0.00139266,-0.491072,0.870802,-0.0234724],[0,-1,-1,0],[9E+09,9E+09,9E+09,9E+09,9E+09,9E+09]],
[[1277.7,64,938.01],[0.00139266,-0.491072,0.870802,-0.0234724],[0,-1,-1,0],[9E+09,9E+09,9E+09,9E+09,9E+09,9E+09]],
[[1278.2,64,938.01],[0.00139266,-0.491072,0.870802,-0.0234724],[0,-1,-1,0],[9E+09,9E+09,9E+09,9E+09,9E+09,9E+09]]
];
CONST robtarget myPath6{21} := [
[[1396.2,31.5,938.01],[0.00139266,-0.491072,0.870802,-0.0234724],[0,-1,-1,0],[9E+09,9E+09,9E+09,9E+09,9E+09,9E+09]],
[[1396.2,31.5,938.01],[0.00139266,-0.491072,0.870802,-0.0234724],[0,-1,-1,0],[9E+09,9E+09,9E+09,9E+09,9E+09,9E+09]],
[[1396.7,31.5,938.01],[0.00139266,-0.491072,0.870802,-0.0234724],[0,-1,-1,0],[9E+09,9E+09,9E+09,9E+09,9E+09,9E+09]],
[[1396.7,31.5,938.01],[0.00139266,-0.491072,0.870802,-0.0234724],[0,-1,-1,0],[9E+09,9E+09,9E+09,9E+09,9E+09,9E+09]],
[[1396.7,31.5,938.01],[0.00139266,-0.491072,0.870802,-0.0234724],[0,-1,-1,0],[9E+09,9E+09,9E+09,9E+09,9E+09,9E+09]],
[[1401.2,35.5,938.01],[0.00139266,-0.491072,0.870802,-0.0234724],[0,-1,-1,0],[9E+09,9E+09,9E+09,9E+09,9E+09,9E+09]],
[[1401.2,41.5,938.01],[0.00139266,-0.491072,0.870802,-0.0234724],[0,-1,-1,0],[9E+09,9E+09,9E+09,9E+09,9E+09,9E+09]],
[[1400.7,42.5,938.01],[0.00139266,-0.491072,0.870802,-0.0234724],[0,-1,-1,0],[9E+09,9E+09,9E+09,9E+09,9E+09,9E+09]],
[[1400.7,42.5,938.01],[0.00139266,-0.491072,0.870802,-0.0234724],[0,-1,-1,0],[9E+09,9E+09,9E+09,9E+09,9E+09,9E+09]],
[[1397.7,44.5,938.01],[0.00139266,-0.491072,0.870802,-0.0234724],[0,-1,-1,0],[9E+09,9E+09,9E+09,9E+09,9E+09,9E+09]],
[[1392.7,43,938.01],[0.00139266,-0.491072,0.870802,-0.0234724],[0,-1,-1,0],[9E+09,9E+09,9E+09,9E+09,9E+09,9E+09]],
[[1392.7,43,938.01],[0.00139266,-0.491072,0.870802,-0.0234724],[0,-1,-1,0],[9E+09,9E+09,9E+09,9E+09,9E+09,9E+09]],
[[1392.7,43,938.01],[0.00139266,-0.491072,0.870802,-0.0234724],[0,-1,-1,0],[9E+09,9E+09,9E+09,9E+09,9E+09,9E+09]],
[[1387.7,38,938.01],[0.00139266,-0.491072,0.870802,-0.0234724],[0,-1,-1,0],[9E+09,9E+09,9E+09,9E+09,9E+09,9E+09]],
[[1387.7,38,938.01],[0.00139266,-0.491072,0.870802,-0.0234724],[0,-1,-1,0],[9E+09,9E+09,9E+09,9E+09,9E+09,9E+09]],
[[1387.7,38,938.01],[0.00139266,-0.491072,0.870802,-0.0234724],[0,-1,-1,0],[9E+09,9E+09,9E+09,9E+09,9E+09,9E+09]],
[[1387.2,37.5,938.01],[0.00139266,-0.491072,0.870802,-0.0234724],[0,-1,-1,0],[9E+09,9E+09,9E+09,9E+09,9E+09,9E+09]],
[[1386.7,36,938.01],[0.00139266,-0.491072,0.870802,-0.0234724],[0,-1,-1,0],[9E+09,9E+09,9E+09,9E+09,9E+09,9E+09]],
[[1387.7,34,938.01],[0.00139266,-0.491072,0.870802,-0.0234724],[0,-1,-1,0],[9E+09,9E+09,9E+09,9E+09,9E+09,9E+09]],
[[1388.2,33.5,938.01],[0.00139266,-0.491072,0.870802,-0.0234724],[0,-1,-1,0],[9E+09,9E+09,9E+09,9E+09,9E+09,9E+09]],
[[1390.2,30.5,938.01],[0.00139266,-0.491072,0.870802,-0.0234724],[0,-1,-1,0],[9E+09,9E+09,9E+09,9E+09,9E+09,9E+09]]
];
CONST robtarget myPath7{96} := [
[[1335.7,1.5,938.01],[0.00139266,-0.491072,0.870802,-0.0234724],[0,-1,-1,0],[9E+09,9E+09,9E+09,9E+09,9E+09,9E+09]],
[[1336.2,2,938.01],[0.00139266,-0.491072,0.870802,-0.0234724],[0,-1,-1,0],[9E+09,9E+09,9E+09,9E+09,9E+09,9E+09]],
[[1339.2,2.5,938.01],[0.00139266,-0.491072,0.870802,-0.0234724],[0,-1,-1,0],[9E+09,9E+09,9E+09,9E+09,9E+09,9E+09]],
[[1340.2,3.5,938.01],[0.00139266,-0.491072,0.870802,-0.0234724],[0,-1,-1,0],[9E+09,9E+09,9E+09,9E+09,9E+09,9E+09]],
[[1342.7,5,938.01],[0.00139266,-0.491072,0.870802,-0.0234724],[0,-1,-1,0],[9E+09,9E+09,9E+09,9E+09,9E+09,9E+09]],
[[1342.7,5,938.01],[0.00139266,-0.491072,0.870802,-0.0234724],[0,-1,-1,0],[9E+09,9E+09,9E+09,9E+09,9E+09,9E+09]],
[[1342.7,5,938.01],[0.00139266,-0.491072,0.870802,-0.0234724],[0,-1,-1,0],[9E+09,9E+09,9E+09,9E+09,9E+09,9E+09]],
[[1342.7,5,938.01],[0.00139266,-0.491072,0.870802,-0.0234724],[0,-1,-1,0],[9E+09,9E+09,9E+09,9E+09,9E+09,9E+09]],
[[1344.7,8,938.01],[0.00139266,-0.491072,0.870802,-0.0234724],[0,-1,-1,0],[9E+09,9E+09,9E+09,9E+09,9E+09,9E+09]],
[[1345.2,9,938.01],[0.00139266,-0.491072,0.870802,-0.0234724],[0,-1,-1,0],[9E+09,9E+09,9E+09,9E+09,9E+09,9E+09]],
[[1345.7,11,938.01],[0.00139266,-0.491072,0.870802,-0.0234724],[0,-1,-1,0],[9E+09,9E+09,9E+09,9E+09,9E+09,9E+09]],
[[1345.7,11,938.01],[0.00139266,-0.491072,0.870802,-0.0234724],[0,-1,-1,0],[9E+09,9E+09,9E+09,9E+09,9E+09,9E+09]],
[[1345.7,11,938.01],[0.00139266,-0.491072,0.870802,-0.0234724],[0,-1,-1,0],[9E+09,9E+09,9E+09,9E+09,9E+09,9E+09]],
[[1345.7,20.5,938.01],[0.00139266,-0.491072,0.870802,-0.0234724],[0,-1,-1,0],[9E+09,9E+09,9E+09,9E+09,9E+09,9E+09]],
[[1345.2,22,938.01],[0.00139266,-0.491072,0.870802,-0.0234724],[0,-1,-1,0],[9E+09,9E+09,9E+09,9E+09,9E+09,9E+09]],
[[1344.7,25.5,938.01],[0.00139266,-0.491072,0.870802,-0.0234724],[0,-1,-1,0],[9E+09,9E+09,9E+09,9E+09,9E+09,9E+09]],
[[1344.2,28,938.01],[0.00139266,-0.491072,0.870802,-0.0234724],[0,-1,-1,0],[9E+09,9E+09,9E+09,9E+09,9E+09,9E+09]],
[[1342.2,37,938.01],[0.00139266,-0.491072,0.870802,-0.0234724],[0,-1,-1,0],[9E+09,9E+09,9E+09,9E+09,9E+09,9E+09]],
[[1341.7,38.5,938.01],[0.00139266,-0.491072,0.870802,-0.0234724],[0,-1,-1,0],[9E+09,9E+09,9E+09,9E+09,9E+09,9E+09]],
[[1341.7,39.5,938.01],[0.00139266,-0.491072,0.870802,-0.0234724],[0,-1,-1,0],[9E+09,9E+09,9E+09,9E+09,9E+09,9E+09]],
[[1340.7,42.5,938.01],[0.00139266,-0.491072,0.870802,-0.0234724],[0,-1,-1,0],[9E+09,9E+09,9E+09,9E+09,9E+09,9E+09]],
[[1340.7,42.5,938.01],[0.00139266,-0.491072,0.870802,-0.0234724],[0,-1,-1,0],[9E+09,9E+09,9E+09,9E+09,9E+09,9E+09]],
[[1340.2,43.5,938.01],[0.00139266,-0.491072,0.870802,-0.0234724],[0,-1,-1,0],[9E+09,9E+09,9E+09,9E+09,9E+09,9E+09]],
[[1340.2,45.5,938.01],[0.00139266,-0.491072,0.870802,-0.0234724],[0,-1,-1,0],[9E+09,9E+09,9E+09,9E+09,9E+09,9E+09]],
[[1339.7,47,938.01],[0.00139266,-0.491072,0.870802,-0.0234724],[0,-1,-1,0],[9E+09,9E+09,9E+09,9E+09,9E+09,9E+09]],
[[1339.7,47,938.01],[0.00139266,-0.491072,0.870802,-0.0234724],[0,-1,-1,0],[9E+09,9E+09,9E+09,9E+09,9E+09,9E+09]],
[[1339.7,47,938.01],[0.00139266,-0.491072,0.870802,-0.0234724],[0,-1,-1,0],[9E+09,9E+09,9E+09,9E+09,9E+09,9E+09]],
[[1338.7,49,938.01],[0.00139266,-0.491072,0.870802,-0.0234724],[0,-1,-1,0],[9E+09,9E+09,9E+09,9E+09,9E+09,9E+09]],
[[1337.7,51.5,938.01],[0.00139266,-0.491072,0.870802,-0.0234724],[0,-1,-1,0],[9E+09,9E+09,9E+09,9E+09,9E+09,9E+09]],
[[1336.7,54,938.01],[0.00139266,-0.491072,0.870802,-0.0234724],[0,-1,-1,0],[9E+09,9E+09,9E+09,9E+09,9E+09,9E+09]],
[[1336.7,54,938.01],[0.00139266,-0.491072,0.870802,-0.0234724],[0,-1,-1,0],[9E+09,9E+09,9E+09,9E+09,9E+09,9E+09]],
[[1336.7,54,938.01],[0.00139266,-0.491072,0.870802,-0.0234724],[0,-1,-1,0],[9E+09,9E+09,9E+09,9E+09,9E+09,9E+09]],
[[1336.7,54.5,938.01],[0.00139266,-0.491072,0.870802,-0.0234724],[0,-1,-1,0],[9E+09,9E+09,9E+09,9E+09,9E+09,9E+09]],
[[1335.7,56,938.01],[0.00139266,-0.491072,0.870802,-0.0234724],[0,-1,-1,0],[9E+09,9E+09,9E+09,9E+09,9E+09,9E+09]],
[[1335.2,57,938.01],[0.00139266,-0.491072,0.870802,-0.0234724],[0,-1,-1,0],[9E+09,9E+09,9E+09,9E+09,9E+09,9E+09]],
[[1334.7,58.5,938.01],[0.00139266,-0.491072,0.870802,-0.0234724],[0,-1,-1,0],[9E+09,9E+09,9E+09,9E+09,9E+09,9E+09]],
[[1334.7,58.5,938.01],[0.00139266,-0.491072,0.870802,-0.0234724],[0,-1,-1,0],[9E+09,9E+09,9E+09,9E+09,9E+09,9E+09]],
[[1334.2,59,938.01],[0.00139266,-0.491072,0.870802,-0.0234724],[0,-1,-1,0],[9E+09,9E+09,9E+09,9E+09,9E+09,9E+09]],
[[1330.2,64.5,938.01],[0.00139266,-0.491072,0.870802,-0.0234724],[0,-1,-1,0],[9E+09,9E+09,9E+09,9E+09,9E+09,9E+09]],
[[1330.2,65,938.01],[0.00139266,-0.491072,0.870802,-0.0234724],[0,-1,-1,0],[9E+09,9E+09,9E+09,9E+09,9E+09,9E+09]],
[[1328.2,67,938.01],[0.00139266,-0.491072,0.870802,-0.0234724],[0,-1,-1,0],[9E+09,9E+09,9E+09,9E+09,9E+09,9E+09]],
[[1327.7,67,938.01],[0.00139266,-0.491072,0.870802,-0.0234724],[0,-1,-1,0],[9E+09,9E+09,9E+09,9E+09,9E+09,9E+09]],
[[1326.7,68,938.01],[0.00139266,-0.491072,0.870802,-0.0234724],[0,-1,-1,0],[9E+09,9E+09,9E+09,9E+09,9E+09,9E+09]],
[[1326.2,68,938.01],[0.00139266,-0.491072,0.870802,-0.0234724],[0,-1,-1,0],[9E+09,9E+09,9E+09,9E+09,9E+09,9E+09]],
[[1323.7,70,938.01],[0.00139266,-0.491072,0.870802,-0.0234724],[0,-1,-1,0],[9E+09,9E+09,9E+09,9E+09,9E+09,9E+09]],
[[1323.7,70,938.01],[0.00139266,-0.491072,0.870802,-0.0234724],[0,-1,-1,0],[9E+09,9E+09,9E+09,9E+09,9E+09,9E+09]],
[[1323.7,70,938.01],[0.00139266,-0.491072,0.870802,-0.0234724],[0,-1,-1,0],[9E+09,9E+09,9E+09,9E+09,9E+09,9E+09]],
[[1320.7,70.5,938.01],[0.00139266,-0.491072,0.870802,-0.0234724],[0,-1,-1,0],[9E+09,9E+09,9E+09,9E+09,9E+09,9E+09]],
[[1317.7,72,938.01],[0.00139266,-0.491072,0.870802,-0.0234724],[0,-1,-1,0],[9E+09,9E+09,9E+09,9E+09,9E+09,9E+09]],
[[1317.7,72,938.01],[0.00139266,-0.491072,0.870802,-0.0234724],[0,-1,-1,0],[9E+09,9E+09,9E+09,9E+09,9E+09,9E+09]],
[[1314.7,71.5,938.01],[0.00139266,-0.491072,0.870802,-0.0234724],[0,-1,-1,0],[9E+09,9E+09,9E+09,9E+09,9E+09,9E+09]],
[[1314.2,71,938.01],[0.00139266,-0.491072,0.870802,-0.0234724],[0,-1,-1,0],[9E+09,9E+09,9E+09,9E+09,9E+09,9E+09]],
[[1310.2,72,938.01],[0.00139266,-0.491072,0.870802,-0.0234724],[0,-1,-1,0],[9E+09,9E+09,9E+09,9E+09,9E+09,9E+09]],
[[1307.2,69.5,938.01],[0.00139266,-0.491072,0.870802,-0.0234724],[0,-1,-1,0],[9E+09,9E+09,9E+09,9E+09,9E+09,9E+09]],
[[1304.2,68.5,938.01],[0.00139266,-0.491072,0.870802,-0.0234724],[0,-1,-1,0],[9E+09,9E+09,9E+09,9E+09,9E+09,9E+09]],
[[1302.2,67,938.01],[0.00139266,-0.491072,0.870802,-0.0234724],[0,-1,-1,0],[9E+09,9E+09,9E+09,9E+09,9E+09,9E+09]],
[[1302.2,67,938.01],[0.00139266,-0.491072,0.870802,-0.0234724],[0,-1,-1,0],[9E+09,9E+09,9E+09,9E+09,9E+09,9E+09]],
[[1296.7,62.5,938.01],[0.00139266,-0.491072,0.870802,-0.0234724],[0,-1,-1,0],[9E+09,9E+09,9E+09,9E+09,9E+09,9E+09]],
[[1295.7,61,938.01],[0.00139266,-0.491072,0.870802,-0.0234724],[0,-1,-1,0],[9E+09,9E+09,9E+09,9E+09,9E+09,9E+09]],
[[1293.7,58,938.01],[0.00139266,-0.491072,0.870802,-0.0234724],[0,-1,-1,0],[9E+09,9E+09,9E+09,9E+09,9E+09,9E+09]],
[[1293.7,58,938.01],[0.00139266,-0.491072,0.870802,-0.0234724],[0,-1,-1,0],[9E+09,9E+09,9E+09,9E+09,9E+09,9E+09]],
[[1293.2,57,938.01],[0.00139266,-0.491072,0.870802,-0.0234724],[0,-1,-1,0],[9E+09,9E+09,9E+09,9E+09,9E+09,9E+09]],
[[1293.2,56.5,938.01],[0.00139266,-0.491072,0.870802,-0.0234724],[0,-1,-1,0],[9E+09,9E+09,9E+09,9E+09,9E+09,9E+09]],
[[1292.7,56,938.01],[0.00139266,-0.491072,0.870802,-0.0234724],[0,-1,-1,0],[9E+09,9E+09,9E+09,9E+09,9E+09,9E+09]],
[[1292.7,42.5,938.01],[0.00139266,-0.491072,0.870802,-0.0234724],[0,-1,-1,0],[9E+09,9E+09,9E+09,9E+09,9E+09,9E+09]],
[[1292.7,42.5,938.01],[0.00139266,-0.491072,0.870802,-0.0234724],[0,-1,-1,0],[9E+09,9E+09,9E+09,9E+09,9E+09,9E+09]],
[[1292.7,42.5,938.01],[0.00139266,-0.491072,0.870802,-0.0234724],[0,-1,-1,0],[9E+09,9E+09,9E+09,9E+09,9E+09,9E+09]],
[[1293.2,41.5,938.01],[0.00139266,-0.491072,0.870802,-0.0234724],[0,-1,-1,0],[9E+09,9E+09,9E+09,9E+09,9E+09,9E+09]],
[[1293.2,41,938.01],[0.00139266,-0.491072,0.870802,-0.0234724],[0,-1,-1,0],[9E+09,9E+09,9E+09,9E+09,9E+09,9E+09]],
[[1293.7,40,938.01],[0.00139266,-0.491072,0.870802,-0.0234724],[0,-1,-1,0],[9E+09,9E+09,9E+09,9E+09,9E+09,9E+09]],
[[1294.2,39,938.01],[0.00139266,-0.491072,0.870802,-0.0234724],[0,-1,-1,0],[9E+09,9E+09,9E+09,9E+09,9E+09,9E+09]],
[[1295.2,36.5,938.01],[0.00139266,-0.491072,0.870802,-0.0234724],[0,-1,-1,0],[9E+09,9E+09,9E+09,9E+09,9E+09,9E+09]],
[[1295.2,36.5,938.01],[0.00139266,-0.491072,0.870802,-0.0234724],[0,-1,-1,0],[9E+09,9E+09,9E+09,9E+09,9E+09,9E+09]],
[[1295.7,35.5,938.01],[0.00139266,-0.491072,0.870802,-0.0234724],[0,-1,-1,0],[9E+09,9E+09,9E+09,9E+09,9E+09,9E+09]],
[[1297.2,32.5,938.01],[0.00139266,-0.491072,0.870802,-0.0234724],[0,-1,-1,0],[9E+09,9E+09,9E+09,9E+09,9E+09,9E+09]],
[[1298.7,30,938.01],[0.00139266,-0.491072,0.870802,-0.0234724],[0,-1,-1,0],[9E+09,9E+09,9E+09,9E+09,9E+09,9E+09]],
[[1298.7,30,938.01],[0.00139266,-0.491072,0.870802,-0.0234724],[0,-1,-1,0],[9E+09,9E+09,9E+09,9E+09,9E+09,9E+09]],
[[1299.2,29.5,938.01],[0.00139266,-0.491072,0.870802,-0.0234724],[0,-1,-1,0],[9E+09,9E+09,9E+09,9E+09,9E+09,9E+09]],
[[1299.7,28.5,938.01],[0.00139266,-0.491072,0.870802,-0.0234724],[0,-1,-1,0],[9E+09,9E+09,9E+09,9E+09,9E+09,9E+09]],
[[1301.7,25.5,938.01],[0.00139266,-0.491072,0.870802,-0.0234724],[0,-1,-1,0],[9E+09,9E+09,9E+09,9E+09,9E+09,9E+09]],
[[1301.7,25.5,938.01],[0.00139266,-0.491072,0.870802,-0.0234724],[0,-1,-1,0],[9E+09,9E+09,9E+09,9E+09,9E+09,9E+09]],
[[1302.2,25,938.01],[0.00139266,-0.491072,0.870802,-0.0234724],[0,-1,-1,0],[9E+09,9E+09,9E+09,9E+09,9E+09,9E+09]],
[[1302.2,25,938.01],[0.00139266,-0.491072,0.870802,-0.0234724],[0,-1,-1,0],[9E+09,9E+09,9E+09,9E+09,9E+09,9E+09]],
[[1303.7,22.5,938.01],[0.00139266,-0.491072,0.870802,-0.0234724],[0,-1,-1,0],[9E+09,9E+09,9E+09,9E+09,9E+09,9E+09]],
[[1303.7,23,938.01],[0.00139266,-0.491072,0.870802,-0.0234724],[0,-1,-1,0],[9E+09,9E+09,9E+09,9E+09,9E+09,9E+09]],
[[1307.2,18.5,938.01],[0.00139266,-0.491072,0.870802,-0.0234724],[0,-1,-1,0],[9E+09,9E+09,9E+09,9E+09,9E+09,9E+09]],
[[1315.2,10,938.01],[0.00139266,-0.491072,0.870802,-0.0234724],[0,-1,-1,0],[9E+09,9E+09,9E+09,9E+09,9E+09,9E+09]],
[[1319.2,7,938.01],[0.00139266,-0.491072,0.870802,-0.0234724],[0,-1,-1,0],[9E+09,9E+09,9E+09,9E+09,9E+09,9E+09]],
[[1319.2,7,938.01],[0.00139266,-0.491072,0.870802,-0.0234724],[0,-1,-1,0],[9E+09,9E+09,9E+09,9E+09,9E+09,9E+09]],
[[1319.7,6.5,938.01],[0.00139266,-0.491072,0.870802,-0.0234724],[0,-1,-1,0],[9E+09,9E+09,9E+09,9E+09,9E+09,9E+09]],
[[1319.7,6.5,938.01],[0.00139266,-0.491072,0.870802,-0.0234724],[0,-1,-1,0],[9E+09,9E+09,9E+09,9E+09,9E+09,9E+09]],
[[1321.2,5.5,938.01],[0.00139266,-0.491072,0.870802,-0.0234724],[0,-1,-1,0],[9E+09,9E+09,9E+09,9E+09,9E+09,9E+09]],
[[1322.2,5,938.01],[0.00139266,-0.491072,0.870802,-0.0234724],[0,-1,-1,0],[9E+09,9E+09,9E+09,9E+09,9E+09,9E+09]],
[[1326.7,3,938.01],[0.00139266,-0.491072,0.870802,-0.0234724],[0,-1,-1,0],[9E+09,9E+09,9E+09,9E+09,9E+09,9E+09]],
[[1327.2,2.5,938.01],[0.00139266,-0.491072,0.870802,-0.0234724],[0,-1,-1,0],[9E+09,9E+09,9E+09,9E+09,9E+09,9E+09]],
[[1327.7,2.5,938.01],[0.00139266,-0.491072,0.870802,-0.0234724],[0,-1,-1,0],[9E+09,9E+09,9E+09,9E+09,9E+09,9E+09]]
];
CONST robtarget myPath8{117} := [
[[1352.2,1,938.01],[0.00139266,-0.491072,0.870802,-0.0234724],[0,-1,-1,0],[9E+09,9E+09,9E+09,9E+09,9E+09,9E+09]],
[[1358.7,1.5,938.01],[0.00139266,-0.491072,0.870802,-0.0234724],[0,-1,-1,0],[9E+09,9E+09,9E+09,9E+09,9E+09,9E+09]],
[[1358.2,1.5,938.01],[0.00139266,-0.491072,0.870802,-0.0234724],[0,-1,-1,0],[9E+09,9E+09,9E+09,9E+09,9E+09,9E+09]],
[[1361.7,2,938.01],[0.00139266,-0.491072,0.870802,-0.0234724],[0,-1,-1,0],[9E+09,9E+09,9E+09,9E+09,9E+09,9E+09]],
[[1362.7,2.5,938.01],[0.00139266,-0.491072,0.870802,-0.0234724],[0,-1,-1,0],[9E+09,9E+09,9E+09,9E+09,9E+09,9E+09]],
[[1365.2,4,938.01],[0.00139266,-0.491072,0.870802,-0.0234724],[0,-1,-1,0],[9E+09,9E+09,9E+09,9E+09,9E+09,9E+09]],
[[1366.2,4.5,938.01],[0.00139266,-0.491072,0.870802,-0.0234724],[0,-1,-1,0],[9E+09,9E+09,9E+09,9E+09,9E+09,9E+09]],
[[1366.7,4.5,938.01],[0.00139266,-0.491072,0.870802,-0.0234724],[0,-1,-1,0],[9E+09,9E+09,9E+09,9E+09,9E+09,9E+09]],
[[1367.2,5,938.01],[0.00139266,-0.491072,0.870802,-0.0234724],[0,-1,-1,0],[9E+09,9E+09,9E+09,9E+09,9E+09,9E+09]],
[[1367.2,5,938.01],[0.00139266,-0.491072,0.870802,-0.0234724],[0,-1,-1,0],[9E+09,9E+09,9E+09,9E+09,9E+09,9E+09]],
[[1370.7,7.5,938.01],[0.00139266,-0.491072,0.870802,-0.0234724],[0,-1,-1,0],[9E+09,9E+09,9E+09,9E+09,9E+09,9E+09]],
[[1371.2,7.5,938.01],[0.00139266,-0.491072,0.870802,-0.0234724],[0,-1,-1,0],[9E+09,9E+09,9E+09,9E+09,9E+09,9E+09]],
[[1376.7,13.5,938.01],[0.00139266,-0.491072,0.870802,-0.0234724],[0,-1,-1,0],[9E+09,9E+09,9E+09,9E+09,9E+09,9E+09]],
[[1377.7,15,938.01],[0.00139266,-0.491072,0.870802,-0.0234724],[0,-1,-1,0],[9E+09,9E+09,9E+09,9E+09,9E+09,9E+09]],
[[1380.7,19,938.01],[0.00139266,-0.491072,0.870802,-0.0234724],[0,-1,-1,0],[9E+09,9E+09,9E+09,9E+09,9E+09,9E+09]],
[[1380.7,19,938.01],[0.00139266,-0.491072,0.870802,-0.0234724],[0,-1,-1,0],[9E+09,9E+09,9E+09,9E+09,9E+09,9E+09]],
[[1382.2,21,938.01],[0.00139266,-0.491072,0.870802,-0.0234724],[0,-1,-1,0],[9E+09,9E+09,9E+09,9E+09,9E+09,9E+09]],
[[1384.7,24.5,938.01],[0.00139266,-0.491072,0.870802,-0.0234724],[0,-1,-1,0],[9E+09,9E+09,9E+09,9E+09,9E+09,9E+09]],
[[1385.2,25,938.01],[0.00139266,-0.491072,0.870802,-0.0234724],[0,-1,-1,0],[9E+09,9E+09,9E+09,9E+09,9E+09,9E+09]],
[[1390.2,30.5,938.01],[0.00139266,-0.491072,0.870802,-0.0234724],[0,-1,-1,0],[9E+09,9E+09,9E+09,9E+09,9E+09,9E+09]],
[[1390.2,30.5,938.01],[0.00139266,-0.491072,0.870802,-0.0234724],[0,-1,-1,0],[9E+09,9E+09,9E+09,9E+09,9E+09,9E+09]],
[[1388.2,33.5,938.01],[0.00139266,-0.491072,0.870802,-0.0234724],[0,-1,-1,0],[9E+09,9E+09,9E+09,9E+09,9E+09,9E+09]],
[[1387.7,34,938.01],[0.00139266,-0.491072,0.870802,-0.0234724],[0,-1,-1,0],[9E+09,9E+09,9E+09,9E+09,9E+09,9E+09]],
[[1386.7,36,938.01],[0.00139266,-0.491072,0.870802,-0.0234724],[0,-1,-1,0],[9E+09,9E+09,9E+09,9E+09,9E+09,9E+09]],
[[1387.2,37.5,938.01],[0.00139266,-0.491072,0.870802,-0.0234724],[0,-1,-1,0],[9E+09,9E+09,9E+09,9E+09,9E+09,9E+09]],
[[1387.7,38,938.01],[0.00139266,-0.491072,0.870802,-0.0234724],[0,-1,-1,0],[9E+09,9E+09,9E+09,9E+09,9E+09,9E+09]],
[[1387.7,38,938.01],[0.00139266,-0.491072,0.870802,-0.0234724],[0,-1,-1,0],[9E+09,9E+09,9E+09,9E+09,9E+09,9E+09]],
[[1387.7,38,938.01],[0.00139266,-0.491072,0.870802,-0.0234724],[0,-1,-1,0],[9E+09,9E+09,9E+09,9E+09,9E+09,9E+09]],
[[1392.7,43,938.01],[0.00139266,-0.491072,0.870802,-0.0234724],[0,-1,-1,0],[9E+09,9E+09,9E+09,9E+09,9E+09,9E+09]],
[[1392.7,43,938.01],[0.00139266,-0.491072,0.870802,-0.0234724],[0,-1,-1,0],[9E+09,9E+09,9E+09,9E+09,9E+09,9E+09]],
[[1395.2,43.5,938.01],[0.00139266,-0.491072,0.870802,-0.0234724],[0,-1,-1,0],[9E+09,9E+09,9E+09,9E+09,9E+09,9E+09]],
[[1398.7,51,938.01],[0.00139266,-0.491072,0.870802,-0.0234724],[0,-1,-1,0],[9E+09,9E+09,9E+09,9E+09,9E+09,9E+09]],
[[1398.2,52.5,938.01],[0.00139266,-0.491072,0.870802,-0.0234724],[0,-1,-1,0],[9E+09,9E+09,9E+09,9E+09,9E+09,9E+09]],
[[1397.7,56,938.01],[0.00139266,-0.491072,0.870802,-0.0234724],[0,-1,-1,0],[9E+09,9E+09,9E+09,9E+09,9E+09,9E+09]],
[[1397.7,56,938.01],[0.00139266,-0.491072,0.870802,-0.0234724],[0,-1,-1,0],[9E+09,9E+09,9E+09,9E+09,9E+09,9E+09]],
[[1396.7,57.5,938.01],[0.00139266,-0.491072,0.870802,-0.0234724],[0,-1,-1,0],[9E+09,9E+09,9E+09,9E+09,9E+09,9E+09]],
[[1395.7,59,938.01],[0.00139266,-0.491072,0.870802,-0.0234724],[0,-1,-1,0],[9E+09,9E+09,9E+09,9E+09,9E+09,9E+09]],
[[1395.7,59.5,938.01],[0.00139266,-0.491072,0.870802,-0.0234724],[0,-1,-1,0],[9E+09,9E+09,9E+09,9E+09,9E+09,9E+09]],
[[1392.7,63.5,938.01],[0.00139266,-0.491072,0.870802,-0.0234724],[0,-1,-1,0],[9E+09,9E+09,9E+09,9E+09,9E+09,9E+09]],
[[1392.7,63.5,938.01],[0.00139266,-0.491072,0.870802,-0.0234724],[0,-1,-1,0],[9E+09,9E+09,9E+09,9E+09,9E+09,9E+09]],
[[1389.2,67,938.01],[0.00139266,-0.491072,0.870802,-0.0234724],[0,-1,-1,0],[9E+09,9E+09,9E+09,9E+09,9E+09,9E+09]],
[[1389.2,67.5,938.01],[0.00139266,-0.491072,0.870802,-0.0234724],[0,-1,-1,0],[9E+09,9E+09,9E+09,9E+09,9E+09,9E+09]],
[[1388.7,67.5,938.01],[0.00139266,-0.491072,0.870802,-0.0234724],[0,-1,-1,0],[9E+09,9E+09,9E+09,9E+09,9E+09,9E+09]],
[[1386.2,69.5,938.01],[0.00139266,-0.491072,0.870802,-0.0234724],[0,-1,-1,0],[9E+09,9E+09,9E+09,9E+09,9E+09,9E+09]],
[[1385.2,70.5,938.01],[0.00139266,-0.491072,0.870802,-0.0234724],[0,-1,-1,0],[9E+09,9E+09,9E+09,9E+09,9E+09,9E+09]],
[[1384.2,71,938.01],[0.00139266,-0.491072,0.870802,-0.0234724],[0,-1,-1,0],[9E+09,9E+09,9E+09,9E+09,9E+09,9E+09]],
[[1384.2,71,938.01],[0.00139266,-0.491072,0.870802,-0.0234724],[0,-1,-1,0],[9E+09,9E+09,9E+09,9E+09,9E+09,9E+09]],
[[1379.2,74,938.01],[0.00139266,-0.491072,0.870802,-0.0234724],[0,-1,-1,0],[9E+09,9E+09,9E+09,9E+09,9E+09,9E+09]],
[[1379.2,74,938.01],[0.00139266,-0.491072,0.870802,-0.0234724],[0,-1,-1,0],[9E+09,9E+09,9E+09,9E+09,9E+09,9E+09]],
[[1377.2,75,938.01],[0.00139266,-0.491072,0.870802,-0.0234724],[0,-1,-1,0],[9E+09,9E+09,9E+09,9E+09,9E+09,9E+09]],
[[1377.2,75,938.01],[0.00139266,-0.491072,0.870802,-0.0234724],[0,-1,-1,0],[9E+09,9E+09,9E+09,9E+09,9E+09,9E+09]],
[[1376.2,75.5,938.01],[0.00139266,-0.491072,0.870802,-0.0234724],[0,-1,-1,0],[9E+09,9E+09,9E+09,9E+09,9E+09,9E+09]],
[[1375.7,76,938.01],[0.00139266,-0.491072,0.870802,-0.0234724],[0,-1,-1,0],[9E+09,9E+09,9E+09,9E+09,9E+09,9E+09]],
[[1375.2,76,938.01],[0.00139266,-0.491072,0.870802,-0.0234724],[0,-1,-1,0],[9E+09,9E+09,9E+09,9E+09,9E+09,9E+09]],
[[1374.7,76,938.01],[0.00139266,-0.491072,0.870802,-0.0234724],[0,-1,-1,0],[9E+09,9E+09,9E+09,9E+09,9E+09,9E+09]],
[[1374.2,76.5,938.01],[0.00139266,-0.491072,0.870802,-0.0234724],[0,-1,-1,0],[9E+09,9E+09,9E+09,9E+09,9E+09,9E+09]],
[[1373.7,76.5,938.01],[0.00139266,-0.491072,0.870802,-0.0234724],[0,-1,-1,0],[9E+09,9E+09,9E+09,9E+09,9E+09,9E+09]],
[[1372.2,77,938.01],[0.00139266,-0.491072,0.870802,-0.0234724],[0,-1,-1,0],[9E+09,9E+09,9E+09,9E+09,9E+09,9E+09]],
[[1371.2,77,938.01],[0.00139266,-0.491072,0.870802,-0.0234724],[0,-1,-1,0],[9E+09,9E+09,9E+09,9E+09,9E+09,9E+09]],
[[1370.7,77.5,938.01],[0.00139266,-0.491072,0.870802,-0.0234724],[0,-1,-1,0],[9E+09,9E+09,9E+09,9E+09,9E+09,9E+09]],
[[1370.2,77.5,938.01],[0.00139266,-0.491072,0.870802,-0.0234724],[0,-1,-1,0],[9E+09,9E+09,9E+09,9E+09,9E+09,9E+09]],
[[1368.2,78,938.01],[0.00139266,-0.491072,0.870802,-0.0234724],[0,-1,-1,0],[9E+09,9E+09,9E+09,9E+09,9E+09,9E+09]],
[[1368.2,78.5,938.01],[0.00139266,-0.491072,0.870802,-0.0234724],[0,-1,-1,0],[9E+09,9E+09,9E+09,9E+09,9E+09,9E+09]],
[[1368.2,78.5,938.01],[0.00139266,-0.491072,0.870802,-0.0234724],[0,-1,-1,0],[9E+09,9E+09,9E+09,9E+09,9E+09,9E+09]],
[[1368.2,78.5,938.01],[0.00139266,-0.491072,0.870802,-0.0234724],[0,-1,-1,0],[9E+09,9E+09,9E+09,9E+09,9E+09,9E+09]],
[[1368.2,78.5,938.01],[0.00139266,-0.491072,0.870802,-0.0234724],[0,-1,-1,0],[9E+09,9E+09,9E+09,9E+09,9E+09,9E+09]],
[[1338.7,79.5,938.01],[0.00139266,-0.491072,0.870802,-0.0234724],[0,-1,-1,0],[9E+09,9E+09,9E+09,9E+09,9E+09,9E+09]],
[[1338.7,79.5,938.01],[0.00139266,-0.491072,0.870802,-0.0234724],[0,-1,-1,0],[9E+09,9E+09,9E+09,9E+09,9E+09,9E+09]],
[[1338.7,79.5,938.01],[0.00139266,-0.491072,0.870802,-0.0234724],[0,-1,-1,0],[9E+09,9E+09,9E+09,9E+09,9E+09,9E+09]],
[[1336.7,78.5,938.01],[0.00139266,-0.491072,0.870802,-0.0234724],[0,-1,-1,0],[9E+09,9E+09,9E+09,9E+09,9E+09,9E+09]],
[[1333.7,77.5,938.01],[0.00139266,-0.491072,0.870802,-0.0234724],[0,-1,-1,0],[9E+09,9E+09,9E+09,9E+09,9E+09,9E+09]],
[[1332.7,77,938.01],[0.00139266,-0.491072,0.870802,-0.0234724],[0,-1,-1,0],[9E+09,9E+09,9E+09,9E+09,9E+09,9E+09]],
[[1330.7,76,938.01],[0.00139266,-0.491072,0.870802,-0.0234724],[0,-1,-1,0],[9E+09,9E+09,9E+09,9E+09,9E+09,9E+09]],
[[1330.7,76,938.01],[0.00139266,-0.491072,0.870802,-0.0234724],[0,-1,-1,0],[9E+09,9E+09,9E+09,9E+09,9E+09,9E+09]],
[[1329.7,75.5,938.01],[0.00139266,-0.491072,0.870802,-0.0234724],[0,-1,-1,0],[9E+09,9E+09,9E+09,9E+09,9E+09,9E+09]],
[[1323.7,70,938.01],[0.00139266,-0.491072,0.870802,-0.0234724],[0,-1,-1,0],[9E+09,9E+09,9E+09,9E+09,9E+09,9E+09]],
[[1326.2,68,938.01],[0.00139266,-0.491072,0.870802,-0.0234724],[0,-1,-1,0],[9E+09,9E+09,9E+09,9E+09,9E+09,9E+09]],
[[1326.7,68,938.01],[0.00139266,-0.491072,0.870802,-0.0234724],[0,-1,-1,0],[9E+09,9E+09,9E+09,9E+09,9E+09,9E+09]],
[[1327.7,67,938.01],[0.00139266,-0.491072,0.870802,-0.0234724],[0,-1,-1,0],[9E+09,9E+09,9E+09,9E+09,9E+09,9E+09]],
[[1328.2,67,938.01],[0.00139266,-0.491072,0.870802,-0.0234724],[0,-1,-1,0],[9E+09,9E+09,9E+09,9E+09,9E+09,9E+09]],
[[1330.2,65,938.01],[0.00139266,-0.491072,0.870802,-0.0234724],[0,-1,-1,0],[9E+09,9E+09,9E+09,9E+09,9E+09,9E+09]],
[[1330.2,64.5,938.01],[0.00139266,-0.491072,0.870802,-0.0234724],[0,-1,-1,0],[9E+09,9E+09,9E+09,9E+09,9E+09,9E+09]],
[[1333.2,60.5,938.01],[0.00139266,-0.491072,0.870802,-0.0234724],[0,-1,-1,0],[9E+09,9E+09,9E+09,9E+09,9E+09,9E+09]],
[[1334.2,59,938.01],[0.00139266,-0.491072,0.870802,-0.0234724],[0,-1,-1,0],[9E+09,9E+09,9E+09,9E+09,9E+09,9E+09]],
[[1334.7,58.5,938.01],[0.00139266,-0.491072,0.870802,-0.0234724],[0,-1,-1,0],[9E+09,9E+09,9E+09,9E+09,9E+09,9E+09]],
[[1334.7,58.5,938.01],[0.00139266,-0.491072,0.870802,-0.0234724],[0,-1,-1,0],[9E+09,9E+09,9E+09,9E+09,9E+09,9E+09]],
[[1335.2,57,938.01],[0.00139266,-0.491072,0.870802,-0.0234724],[0,-1,-1,0],[9E+09,9E+09,9E+09,9E+09,9E+09,9E+09]],
[[1335.7,56,938.01],[0.00139266,-0.491072,0.870802,-0.0234724],[0,-1,-1,0],[9E+09,9E+09,9E+09,9E+09,9E+09,9E+09]],
[[1336.7,54.5,938.01],[0.00139266,-0.491072,0.870802,-0.0234724],[0,-1,-1,0],[9E+09,9E+09,9E+09,9E+09,9E+09,9E+09]],
[[1336.7,54,938.01],[0.00139266,-0.491072,0.870802,-0.0234724],[0,-1,-1,0],[9E+09,9E+09,9E+09,9E+09,9E+09,9E+09]],
[[1336.7,54,938.01],[0.00139266,-0.491072,0.870802,-0.0234724],[0,-1,-1,0],[9E+09,9E+09,9E+09,9E+09,9E+09,9E+09]],
[[1336.7,54,938.01],[0.00139266,-0.491072,0.870802,-0.0234724],[0,-1,-1,0],[9E+09,9E+09,9E+09,9E+09,9E+09,9E+09]],
[[1338.2,50.5,938.01],[0.00139266,-0.491072,0.870802,-0.0234724],[0,-1,-1,0],[9E+09,9E+09,9E+09,9E+09,9E+09,9E+09]],
[[1338.7,49,938.01],[0.00139266,-0.491072,0.870802,-0.0234724],[0,-1,-1,0],[9E+09,9E+09,9E+09,9E+09,9E+09,9E+09]],
[[1338.7,49,938.01],[0.00139266,-0.491072,0.870802,-0.0234724],[0,-1,-1,0],[9E+09,9E+09,9E+09,9E+09,9E+09,9E+09]],
[[1339.7,47,938.01],[0.00139266,-0.491072,0.870802,-0.0234724],[0,-1,-1,0],[9E+09,9E+09,9E+09,9E+09,9E+09,9E+09]],
[[1339.7,47,938.01],[0.00139266,-0.491072,0.870802,-0.0234724],[0,-1,-1,0],[9E+09,9E+09,9E+09,9E+09,9E+09,9E+09]],
[[1340.2,45.5,938.01],[0.00139266,-0.491072,0.870802,-0.0234724],[0,-1,-1,0],[9E+09,9E+09,9E+09,9E+09,9E+09,9E+09]],
[[1340.2,43.5,938.01],[0.00139266,-0.491072,0.870802,-0.0234724],[0,-1,-1,0],[9E+09,9E+09,9E+09,9E+09,9E+09,9E+09]],
[[1340.7,42.5,938.01],[0.00139266,-0.491072,0.870802,-0.0234724],[0,-1,-1,0],[9E+09,9E+09,9E+09,9E+09,9E+09,9E+09]],
[[1340.7,42.5,938.01],[0.00139266,-0.491072,0.870802,-0.0234724],[0,-1,-1,0],[9E+09,9E+09,9E+09,9E+09,9E+09,9E+09]],
[[1341.7,39.5,938.01],[0.00139266,-0.491072,0.870802,-0.0234724],[0,-1,-1,0],[9E+09,9E+09,9E+09,9E+09,9E+09,9E+09]],
[[1341.7,38.5,938.01],[0.00139266,-0.491072,0.870802,-0.0234724],[0,-1,-1,0],[9E+09,9E+09,9E+09,9E+09,9E+09,9E+09]],
[[1342.2,37,938.01],[0.00139266,-0.491072,0.870802,-0.0234724],[0,-1,-1,0],[9E+09,9E+09,9E+09,9E+09,9E+09,9E+09]],
[[1343.2,31.5,938.01],[0.00139266,-0.491072,0.870802,-0.0234724],[0,-1,-1,0],[9E+09,9E+09,9E+09,9E+09,9E+09,9E+09]],
[[1344.7,25.5,938.01],[0.00139266,-0.491072,0.870802,-0.0234724],[0,-1,-1,0],[9E+09,9E+09,9E+09,9E+09,9E+09,9E+09]],
[[1345.2,22,938.01],[0.00139266,-0.491072,0.870802,-0.0234724],[0,-1,-1,0],[9E+09,9E+09,9E+09,9E+09,9E+09,9E+09]],
[[1345.7,20.5,938.01],[0.00139266,-0.491072,0.870802,-0.0234724],[0,-1,-1,0],[9E+09,9E+09,9E+09,9E+09,9E+09,9E+09]],
[[1345.7,11,938.01],[0.00139266,-0.491072,0.870802,-0.0234724],[0,-1,-1,0],[9E+09,9E+09,9E+09,9E+09,9E+09,9E+09]],
[[1345.7,11,938.01],[0.00139266,-0.491072,0.870802,-0.0234724],[0,-1,-1,0],[9E+09,9E+09,9E+09,9E+09,9E+09,9E+09]],
[[1345.7,11,938.01],[0.00139266,-0.491072,0.870802,-0.0234724],[0,-1,-1,0],[9E+09,9E+09,9E+09,9E+09,9E+09,9E+09]],
[[1345.2,9,938.01],[0.00139266,-0.491072,0.870802,-0.0234724],[0,-1,-1,0],[9E+09,9E+09,9E+09,9E+09,9E+09,9E+09]],
[[1344.7,8,938.01],[0.00139266,-0.491072,0.870802,-0.0234724],[0,-1,-1,0],[9E+09,9E+09,9E+09,9E+09,9E+09,9E+09]],
[[1342.7,5,938.01],[0.00139266,-0.491072,0.870802,-0.0234724],[0,-1,-1,0],[9E+09,9E+09,9E+09,9E+09,9E+09,9E+09]],
[[1342.7,5,938.01],[0.00139266,-0.491072,0.870802,-0.0234724],[0,-1,-1,0],[9E+09,9E+09,9E+09,9E+09,9E+09,9E+09]],
[[1345.7,3,938.01],[0.00139266,-0.491072,0.870802,-0.0234724],[0,-1,-1,0],[9E+09,9E+09,9E+09,9E+09,9E+09,9E+09]],
[[1346.2,3,938.01],[0.00139266,-0.491072,0.870802,-0.0234724],[0,-1,-1,0],[9E+09,9E+09,9E+09,9E+09,9E+09,9E+09]]
];
CONST robtarget myPath9{9} := [
[[1362.2,70.5,938.01],[0.00139266,-0.491072,0.870802,-0.0234724],[0,-1,-1,0],[9E+09,9E+09,9E+09,9E+09,9E+09,9E+09]],
[[1362.2,70.5,938.01],[0.00139266,-0.491072,0.870802,-0.0234724],[0,-1,-1,0],[9E+09,9E+09,9E+09,9E+09,9E+09,9E+09]],
[[1367.7,70.5,938.01],[0.00139266,-0.491072,0.870802,-0.0234724],[0,-1,-1,0],[9E+09,9E+09,9E+09,9E+09,9E+09,9E+09]],
[[1369.7,68,938.01],[0.00139266,-0.491072,0.870802,-0.0234724],[0,-1,-1,0],[9E+09,9E+09,9E+09,9E+09,9E+09,9E+09]],
[[1369.7,68,938.01],[0.00139266,-0.491072,0.870802,-0.0234724],[0,-1,-1,0],[9E+09,9E+09,9E+09,9E+09,9E+09,9E+09]],
[[1369.7,68,938.01],[0.00139266,-0.491072,0.870802,-0.0234724],[0,-1,-1,0],[9E+09,9E+09,9E+09,9E+09,9E+09,9E+09]],
[[1367.7,70.5,938.01],[0.00139266,-0.491072,0.870802,-0.0234724],[0,-1,-1,0],[9E+09,9E+09,9E+09,9E+09,9E+09,9E+09]],
[[1362.2,70.5,938.01],[0.00139266,-0.491072,0.870802,-0.0234724],[0,-1,-1,0],[9E+09,9E+09,9E+09,9E+09,9E+09,9E+09]],
[[1362.2,70.5,938.01],[0.00139266,-0.491072,0.870802,-0.0234724],[0,-1,-1,0],[9E+09,9E+09,9E+09,9E+09,9E+09,9E+09]]
];
CONST robtarget myPath10{21} := [
[[1361.7,28,938.01],[0.00139266,-0.491072,0.870802,-0.0234724],[0,-1,-1,0],[9E+09,9E+09,9E+09,9E+09,9E+09,9E+09]],
[[1361.7,28,938.01],[0.00139266,-0.491072,0.870802,-0.0234724],[0,-1,-1,0],[9E+09,9E+09,9E+09,9E+09,9E+09,9E+09]],
[[1356.7,32.5,938.01],[0.00139266,-0.491072,0.870802,-0.0234724],[0,-1,-1,0],[9E+09,9E+09,9E+09,9E+09,9E+09,9E+09]],
[[1356.7,32.5,938.01],[0.00139266,-0.491072,0.870802,-0.0234724],[0,-1,-1,0],[9E+09,9E+09,9E+09,9E+09,9E+09,9E+09]],
[[1355.2,36,938.01],[0.00139266,-0.491072,0.870802,-0.0234724],[0,-1,-1,0],[9E+09,9E+09,9E+09,9E+09,9E+09,9E+09]],
[[1358.7,40.5,938.01],[0.00139266,-0.491072,0.870802,-0.0234724],[0,-1,-1,0],[9E+09,9E+09,9E+09,9E+09,9E+09,9E+09]],
[[1359.2,40.5,938.01],[0.00139266,-0.491072,0.870802,-0.0234724],[0,-1,-1,0],[9E+09,9E+09,9E+09,9E+09,9E+09,9E+09]],
[[1362.2,41.5,938.01],[0.00139266,-0.491072,0.870802,-0.0234724],[0,-1,-1,0],[9E+09,9E+09,9E+09,9E+09,9E+09,9E+09]],
[[1368.2,41,938.01],[0.00139266,-0.491072,0.870802,-0.0234724],[0,-1,-1,0],[9E+09,9E+09,9E+09,9E+09,9E+09,9E+09]],
[[1368.2,41,938.01],[0.00139266,-0.491072,0.870802,-0.0234724],[0,-1,-1,0],[9E+09,9E+09,9E+09,9E+09,9E+09,9E+09]],
[[1368.2,41,938.01],[0.00139266,-0.491072,0.870802,-0.0234724],[0,-1,-1,0],[9E+09,9E+09,9E+09,9E+09,9E+09,9E+09]],
[[1368.2,41,938.01],[0.00139266,-0.491072,0.870802,-0.0234724],[0,-1,-1,0],[9E+09,9E+09,9E+09,9E+09,9E+09,9E+09]],
[[1368.2,41,938.01],[0.00139266,-0.491072,0.870802,-0.0234724],[0,-1,-1,0],[9E+09,9E+09,9E+09,9E+09,9E+09,9E+09]],
[[1371.7,37.5,938.01],[0.00139266,-0.491072,0.870802,-0.0234724],[0,-1,-1,0],[9E+09,9E+09,9E+09,9E+09,9E+09,9E+09]],
[[1371.7,37.5,938.01],[0.00139266,-0.491072,0.870802,-0.0234724],[0,-1,-1,0],[9E+09,9E+09,9E+09,9E+09,9E+09,9E+09]],
[[1372.2,36.5,938.01],[0.00139266,-0.491072,0.870802,-0.0234724],[0,-1,-1,0],[9E+09,9E+09,9E+09,9E+09,9E+09,9E+09]],
[[1372.2,34.5,938.01],[0.00139266,-0.491072,0.870802,-0.0234724],[0,-1,-1,0],[9E+09,9E+09,9E+09,9E+09,9E+09,9E+09]],
[[1371.2,32.5,938.01],[0.00139266,-0.491072,0.870802,-0.0234724],[0,-1,-1,0],[9E+09,9E+09,9E+09,9E+09,9E+09,9E+09]],
[[1371.2,32.5,938.01],[0.00139266,-0.491072,0.870802,-0.0234724],[0,-1,-1,0],[9E+09,9E+09,9E+09,9E+09,9E+09,9E+09]],
[[1368.7,30,938.01],[0.00139266,-0.491072,0.870802,-0.0234724],[0,-1,-1,0],[9E+09,9E+09,9E+09,9E+09,9E+09,9E+09]],
[[1365.2,28,938.01],[0.00139266,-0.491072,0.870802,-0.0234724],[0,-1,-1,0],[9E+09,9E+09,9E+09,9E+09,9E+09,9E+09]]
];
CONST robtarget myPath11{17} := [
[[1368.7,30,938.01],[0.00139266,-0.491072,0.870802,-0.0234724],[0,-1,-1,0],[9E+09,9E+09,9E+09,9E+09,9E+09,9E+09]],
[[1368.7,30,938.01],[0.00139266,-0.491072,0.870802,-0.0234724],[0,-1,-1,0],[9E+09,9E+09,9E+09,9E+09,9E+09,9E+09]],
[[1371.7,33,938.01],[0.00139266,-0.491072,0.870802,-0.0234724],[0,-1,-1,0],[9E+09,9E+09,9E+09,9E+09,9E+09,9E+09]],
[[1372.2,34.5,938.01],[0.00139266,-0.491072,0.870802,-0.0234724],[0,-1,-1,0],[9E+09,9E+09,9E+09,9E+09,9E+09,9E+09]],
[[1372.2,36.5,938.01],[0.00139266,-0.491072,0.870802,-0.0234724],[0,-1,-1,0],[9E+09,9E+09,9E+09,9E+09,9E+09,9E+09]],
[[1371.7,37.5,938.01],[0.00139266,-0.491072,0.870802,-0.0234724],[0,-1,-1,0],[9E+09,9E+09,9E+09,9E+09,9E+09,9E+09]],
[[1371.7,37.5,938.01],[0.00139266,-0.491072,0.870802,-0.0234724],[0,-1,-1,0],[9E+09,9E+09,9E+09,9E+09,9E+09,9E+09]],
[[1368.2,41,938.01],[0.00139266,-0.491072,0.870802,-0.0234724],[0,-1,-1,0],[9E+09,9E+09,9E+09,9E+09,9E+09,9E+09]],
[[1368.2,41,938.01],[0.00139266,-0.491072,0.870802,-0.0234724],[0,-1,-1,0],[9E+09,9E+09,9E+09,9E+09,9E+09,9E+09]],
[[1361.7,41.5,938.01],[0.00139266,-0.491072,0.870802,-0.0234724],[0,-1,-1,0],[9E+09,9E+09,9E+09,9E+09,9E+09,9E+09]],
[[1361.2,38.5,938.01],[0.00139266,-0.491072,0.870802,-0.0234724],[0,-1,-1,0],[9E+09,9E+09,9E+09,9E+09,9E+09,9E+09]],
[[1361.7,35,938.01],[0.00139266,-0.491072,0.870802,-0.0234724],[0,-1,-1,0],[9E+09,9E+09,9E+09,9E+09,9E+09,9E+09]],
[[1361.7,35,938.01],[0.00139266,-0.491072,0.870802,-0.0234724],[0,-1,-1,0],[9E+09,9E+09,9E+09,9E+09,9E+09,9E+09]],
[[1364.2,32,938.01],[0.00139266,-0.491072,0.870802,-0.0234724],[0,-1,-1,0],[9E+09,9E+09,9E+09,9E+09,9E+09,9E+09]],
[[1364.7,32,938.01],[0.00139266,-0.491072,0.870802,-0.0234724],[0,-1,-1,0],[9E+09,9E+09,9E+09,9E+09,9E+09,9E+09]],
[[1365.7,31,938.01],[0.00139266,-0.491072,0.870802,-0.0234724],[0,-1,-1,0],[9E+09,9E+09,9E+09,9E+09,9E+09,9E+09]],
[[1366.2,31,938.01],[0.00139266,-0.491072,0.870802,-0.0234724],[0,-1,-1,0],[9E+09,9E+09,9E+09,9E+09,9E+09,9E+09]]
];
CONST robtarget myPath12{18} := [
[[1364.7,27.5,938.01],[0.00139266,-0.491072,0.870802,-0.0234724],[0,-1,-1,0],[9E+09,9E+09,9E+09,9E+09,9E+09,9E+09]],
[[1365.2,28,938.01],[0.00139266,-0.491072,0.870802,-0.0234724],[0,-1,-1,0],[9E+09,9E+09,9E+09,9E+09,9E+09,9E+09]],
[[1368.7,30,938.01],[0.00139266,-0.491072,0.870802,-0.0234724],[0,-1,-1,0],[9E+09,9E+09,9E+09,9E+09,9E+09,9E+09]],
[[1366.2,30.5,938.01],[0.00139266,-0.491072,0.870802,-0.0234724],[0,-1,-1,0],[9E+09,9E+09,9E+09,9E+09,9E+09,9E+09]],
[[1365.2,31.5,938.01],[0.00139266,-0.491072,0.870802,-0.0234724],[0,-1,-1,0],[9E+09,9E+09,9E+09,9E+09,9E+09,9E+09]],
[[1364.7,31.5,938.01],[0.00139266,-0.491072,0.870802,-0.0234724],[0,-1,-1,0],[9E+09,9E+09,9E+09,9E+09,9E+09,9E+09]],
[[1364.2,32,938.01],[0.00139266,-0.491072,0.870802,-0.0234724],[0,-1,-1,0],[9E+09,9E+09,9E+09,9E+09,9E+09,9E+09]],
[[1363.7,32,938.01],[0.00139266,-0.491072,0.870802,-0.0234724],[0,-1,-1,0],[9E+09,9E+09,9E+09,9E+09,9E+09,9E+09]],
[[1361.7,35,938.01],[0.00139266,-0.491072,0.870802,-0.0234724],[0,-1,-1,0],[9E+09,9E+09,9E+09,9E+09,9E+09,9E+09]],
[[1361.7,35,938.01],[0.00139266,-0.491072,0.870802,-0.0234724],[0,-1,-1,0],[9E+09,9E+09,9E+09,9E+09,9E+09,9E+09]],
[[1361.7,35,938.01],[0.00139266,-0.491072,0.870802,-0.0234724],[0,-1,-1,0],[9E+09,9E+09,9E+09,9E+09,9E+09,9E+09]],
[[1359.2,40.5,938.01],[0.00139266,-0.491072,0.870802,-0.0234724],[0,-1,-1,0],[9E+09,9E+09,9E+09,9E+09,9E+09,9E+09]],
[[1358.7,40.5,938.01],[0.00139266,-0.491072,0.870802,-0.0234724],[0,-1,-1,0],[9E+09,9E+09,9E+09,9E+09,9E+09,9E+09]],
[[1355.2,36,938.01],[0.00139266,-0.491072,0.870802,-0.0234724],[0,-1,-1,0],[9E+09,9E+09,9E+09,9E+09,9E+09,9E+09]],
[[1355.2,36,938.01],[0.00139266,-0.491072,0.870802,-0.0234724],[0,-1,-1,0],[9E+09,9E+09,9E+09,9E+09,9E+09,9E+09]],
[[1356.7,32.5,938.01],[0.00139266,-0.491072,0.870802,-0.0234724],[0,-1,-1,0],[9E+09,9E+09,9E+09,9E+09,9E+09,9E+09]],
[[1361.7,28,938.01],[0.00139266,-0.491072,0.870802,-0.0234724],[0,-1,-1,0],[9E+09,9E+09,9E+09,9E+09,9E+09,9E+09]],
[[1361.7,28,938.01],[0.00139266,-0.491072,0.870802,-0.0234724],[0,-1,-1,0],[9E+09,9E+09,9E+09,9E+09,9E+09,9E+09]]
];

    PROC draw_path(robtarget arr{*})
        SetDO SETPEN, 0;
        MoveL arr{1}, v50, z5, AW_Gun;
        WaitTime 1;
        SetDO SETPEN, 1;
        FOR i FROM 2 TO Dim(arr, 1) DO
            MoveL arr{i}, v50, z5, AW_Gun;
        ENDFOR
        WaitTime 0.5;
    ENDPROC


    PROC main()
        SetDO SETPEN, 0;
        WaitTime 1;
        draw_path(myPath0);
        WaitTime 0.5;
        draw_path(myPath1);
        WaitTime 0.5;
        draw_path(myPath2);
        WaitTime 0.5;
        draw_path(myPath3);
        WaitTime 0.5;
        draw_path(myPath4);
        WaitTime 0.5;
        draw_path(myPath5);
        WaitTime 0.5;
        draw_path(myPath6);
        WaitTime 0.5;
        draw_path(myPath7);
        WaitTime 0.5;
        draw_path(myPath8);
        WaitTime 0.5;
        draw_path(myPath9);
        WaitTime 0.5;
        draw_path(myPath10);
        WaitTime 0.5;
        draw_path(myPath11);
        WaitTime 0.5;
        draw_path(myPath12);
        WaitTime 0.5;
        SetDO SETPEN, 0;
    ENDPROC

ENDMODULE
